LIN {X 0,Y 186.337,Z 566.167,A -85,B 0,C 180,E1 -25155.389,E2 -25155.389} C_VEL
LIN {X 0,Y 191.242,Z 552.199,A -85,B 0,C 180,E1 -25156.919,E2 -25156.919} C_VEL
LIN {X 0,Y 195.713,Z 537.266,A -85,B 0,C 180,E1 -25158.17,E2 -25158.17} C_VEL
LIN {X 0,Y 199.579,Z 520.667,A -85,B 0,C 180,E1 -25159.209,E2 -25159.209} C_VEL
LIN {X 0,Y 202.453,Z 503.675,A -85,B 0,C 180,E1 -25159.932,E2 -25159.932} C_VEL
LIN {X 0,Y 204.963,Z 478.891,A -85,B 0,C 180,E1 -25160.624,E2 -25160.624} C_VEL
LIN {X 0,Y 210.105,Z 419.825,A -85,B 0,C 180,E1 -25162.198,E2 -25162.198} C_VEL
LIN {X 0,Y 205.857,Z 410.908,A -85,B 0,C 180,E1 -25164.939,E2 -25164.939} C_VEL
LIN {X 0,Y 201.466,Z 402.465,A -85,B 0,C 180,E1 -25168.126,E2 -25168.126} C_VEL
LIN {X 0,Y 197.062,Z 394.449,A -85,B 0,C 180,E1 -25171.873,E2 -25171.873} C_VEL
LIN {X 0,Y 194.207,Z 389.891,A -85,B 0,C 180,E1 -25174.726,E2 -25174.726} C_VEL
LIN {X 0,Y 192.533,Z 387.216,A -85,B 0,C 180,E1 -25176.669,E2 -25176.669} C_VEL
LIN {X 0,Y 190.23,Z 383.452,A -85,B 0,C 180,E1 -25179.848,E2 -25179.848} C_VEL
LIN {X 0,Y 188.062,Z 379.924,A -85,B 0,C 180,E1 -25183.828,E2 -25183.828} C_VEL
LIN {X 0,Y 187.657,Z 379.206,A -85,B 0,C 180,E1 -25184.801,E2 -25184.801} C_VEL
LIN {X 0,Y 185.966,Z 376.838,A -85,B 0,C 180,E1 -25192.422,E2 -25192.422} C_VEL
LIN {X 0,Y 186.444,Z 377.313,A -85,B 0,C 180,E1 -25197.839,E2 -25197.839} C_VEL
LIN {X 0,Y 188.185,Z 379.6,A -85,B 0,C 180,E1 -25202.937,E2 -25202.937} C_VEL
LIN {X 0,Y 190.422,Z 383.385,A -85,B 0,C 180,E1 -25207.007,E2 -25207.007} C_VEL
LIN {X 0,Y 193.373,Z 388.362,A -85,B 0,C 180,E1 -25210.924,E2 -25210.924} C_VEL
LIN {X 0,Y 196.208,Z 393.162,A -85,B 0,C 180,E1 -25213.941,E2 -25213.941} C_VEL
LIN {X 0,Y 199.236,Z 398.22,A -85,B 0,C 180,E1 -25216.662,E2 -25216.662} C_VEL
LIN {X 0,Y 203.737,Z 406.658,A -85,B 0,C 180,E1 -25220.178,E2 -25220.178} C_VEL
LIN {X 0,Y 206.831,Z 412.903,A -85,B 0,C 180,E1 -25222.329,E2 -25222.329} C_VEL
LIN {X 0,Y 210.145,Z 421.82,A -85,B 0,C 180,E1 -25224.569,E2 -25224.569} C_VEL
LIN {X 0,Y 202.457,Z 507.175,A -85,B 0,C 180,E1 -25226.824,E2 -25226.824} C_VEL
LIN {X 0,Y 199.785,Z 523.819,A -85,B 0,C 180,E1 -25227.486,E2 -25227.486} C_VEL
LIN {X 0,Y 196.167,Z 539.714,A -85,B 0,C 180,E1 -25228.359,E2 -25228.359} C_VEL
LIN {X 0,Y 191.397,Z 555.971,A -85,B 0,C 180,E1 -25229.566,E2 -25229.566} C_VEL
LIN {X 0,Y 186.522,Z 570.12,A -85,B 0,C 180,E1 -25230.996,E2 -25230.996} C_VEL
LIN {X 0,Y 180.009,Z 585.472,A -85,B 0,C 180,E1 -25232.924,E2 -25232.924} C_VEL
LIN {X 0,Y 177.704,Z 590.398,A -85,B 0,C 180,E1 -25233.681,E2 -25233.681} C_VEL
LIN {X 0,Y 174.983,Z 595.274,A -85,B 0,C 180,E1 -25234.341,E2 -25234.341} C_VEL
LIN {X 0,Y 164.141,Z 608.926,A -85,B 0,C 180,E1 -25235.695,E2 -25235.695} C_VEL
LIN {X 0,Y 160.851,Z 613.295,A -85,B 0,C 180,E1 -25236.464,E2 -25236.464} C_VEL
LIN {X 0,Y 159.931,Z 614.738,A -85,B 0,C 180,E1 -25236.807,E2 -25236.807} C_VEL
LIN {X 0,Y 152.687,Z 626.22,A -85,B 0,C 180,E1 -25240.119,E2 -25240.119} C_VEL
LIN {X 0,Y 144.962,Z 637.569,A -85,B 0,C 180,E1 -25244.349,E2 -25244.349} C_VEL
LIN {X 0,Y 138.444,Z 646.665,A -85,B 0,C 180,E1 -25248.706,E2 -25248.706} C_VEL
LIN {X 0,Y 132.088,Z 655.399,A -85,B 0,C 180,E1 -25254.178,E2 -25254.178} C_VEL
LIN {X 0,Y 126.943,Z 662.627,A -85,B 0,C 180,E1 -25260.115,E2 -25260.115} C_VEL
LIN {X 0,Y 123.111,Z 668.58,A -85,B 0,C 180,E1 -25266.447,E2 -25266.447} C_VEL
LIN {X 0,Y 120.642,Z 673.309,A -85,B 0,C 180,E1 -25273.066,E2 -25273.066} C_VEL
LIN {X 0,Y 119.404,Z 676.892,A -85,B 0,C 180,E1 -25279.83,E2 -25279.83} C_VEL
LIN {X 0,Y 119.27,Z 679.447,A -85,B 0,C 180,E1 -25286.622,E2 -25286.622} C_VEL
LIN {X 0,Y 119.387,Z 680.288,A -85,B 0,C 180,E1 -25290,E2 -25290} C_VEL
LIN {X 0,Y 119.192,Z 681.267,A -85,B 0,C 180,E1 -25296.773,E2 -25296.773} C_VEL
LIN {X 0,Y 119.91,Z 681.236,A -85,B 0,C 180,E1 -25303.559,E2 -25303.559} C_VEL
LIN {X 0,Y 121.953,Z 680.336,A -85,B 0,C 180,E1 -25310.229,E2 -25310.229} C_VEL
LIN {X 0,Y 125.364,Z 678.424,A -85,B 0,C 180,E1 -25316.647,E2 -25316.647} C_VEL
LIN {X 0,Y 130.22,Z 675.643,A -85,B 0,C 180,E1 -25322.664,E2 -25322.664} C_VEL
LIN {X 0,Y 138.009,Z 670.706,A -85,B 0,C 180,E1 -25329.536,E2 -25329.536} C_VEL
LIN {X 0,Y 147.62,Z 664.098,A -85,B 0,C 180,E1 -25335.573,E2 -25335.573} C_VEL
LIN {X 0,Y 156.377,Z 657.468,A -85,B 0,C 180,E1 -25339.821,E2 -25339.821} C_VEL
LIN {X 0,Y 166.999,Z 648.604,A -85,B 0,C 180,E1 -25344.005,E2 -25344.005} C_VEL
LIN {X 0,Y 177.411,Z 638.938,A -85,B 0,C 180,E1 -25347.331,E2 -25347.331} C_VEL
LIN {X 0,Y 186.913,Z 629.099,A -85,B 0,C 180,E1 -25349.861,E2 -25349.861} C_VEL
LIN {X 0,Y 196.077,Z 618.371,A -85,B 0,C 180,E1 -25352.022,E2 -25352.022} C_VEL
LIN {X 0,Y 204.663,Z 607.189,A -85,B 0,C 180,E1 -25353.782,E2 -25353.782} C_VEL
LIN {X 0,Y 213.545,Z 593.939,A -85,B 0,C 180,E1 -25355.391,E2 -25355.391} C_VEL
LIN {X 0,Y 221.834,Z 579.493,A -85,B 0,C 180,E1 -25356.746,E2 -25356.746} C_VEL
LIN {X 0,Y 228.693,Z 565.379,A -85,B 0,C 180,E1 -25357.786,E2 -25357.786} C_VEL
LIN {X 0,Y 234.898,Z 550.175,A -85,B 0,C 180,E1 -25358.63,E2 -25358.63} C_VEL
LIN {X 0,Y 239.98,Z 534.664,A -85,B 0,C 180,E1 -25359.279,E2 -25359.279} C_VEL
LIN {X 0,Y 244.021,Z 518.311,A -85,B 0,C 180,E1 -25359.771,E2 -25359.771} C_VEL
LIN {X 0,Y 246.768,Z 501.84,A -85,B 0,C 180,E1 -25360.179,E2 -25360.179} C_VEL
LIN {X 0,Y 251.671,Z 457.038,A -85,B 0,C 180,E1 -25361.057,E2 -25361.057} C_VEL
LIN {X 0,Y 250.215,Z 453.342,A -85,B 0,C 180,E1 -25363.107,E2 -25363.107} C_VEL
LIN {X 0,Y 248.725,Z 450.046,A -85,B 0,C 180,E1 -25365.709,E2 -25365.709} C_VEL
LIN {X 0,Y 247.616,Z 447.275,A -85,B 0,C 180,E1 -25368.541,E2 -25368.541} C_VEL
LIN {X 0,Y 246.778,Z 445.427,A -85,B 0,C 180,E1 -25373.46,E2 -25373.46} C_VEL
LIN {X 0,Y 247.261,Z 446.348,A -85,B 0,C 180,E1 -25377.569,E2 -25377.569} C_VEL
LIN {X 0,Y 247.838,Z 447.378,A -85,B 0,C 180,E1 -25379.455,E2 -25379.455} C_VEL
LIN {X 0,Y 249.181,Z 450.878,A -85,B 0,C 180,E1 -25382.582,E2 -25382.582} C_VEL
LIN {X 0,Y 250.647,Z 454.357,A -85,B 0,C 180,E1 -25384.977,E2 -25384.977} C_VEL
LIN {X 0,Y 251.649,Z 456.664,A -85,B 0,C 180,E1 -25386.321,E2 -25386.321} C_VEL
LIN {X 0,Y 246.521,Z 502.914,A -85,B 0,C 180,E1 -25387.271,E2 -25387.271} C_VEL
LIN {X 0,Y 243.089,Z 520.449,A -85,B 0,C 180,E1 -25387.703,E2 -25387.703} C_VEL
LIN {X 0,Y 239.582,Z 533.686,A -85,B 0,C 180,E1 -25388.23,E2 -25388.23} C_VEL
LIN {X 0,Y 234.385,Z 549.286,A -85,B 0,C 180,E1 -25389.021,E2 -25389.021} C_VEL
LIN {X 0,Y 228.35,Z 563.869,A -85,B 0,C 180,E1 -25389.976,E2 -25389.976} C_VEL
LIN {X 0,Y 221.177,Z 578.22,A -85,B 0,C 180,E1 -25391.166,E2 -25391.166} C_VEL
LIN {X 0,Y 213.319,Z 591.621,A -85,B 0,C 180,E1 -25392.57,E2 -25392.57} C_VEL
LIN {X 0,Y 204.35,Z 604.831,A -85,B 0,C 180,E1 -25394.347,E2 -25394.347} C_VEL
LIN {X 0,Y 194.601,Z 617.303,A -85,B 0,C 180,E1 -25396.523,E2 -25396.523} C_VEL
LIN {X 0,Y 184.196,Z 628.903,A -85,B 0,C 180,E1 -25399.206,E2 -25399.206} C_VEL
LIN {X 0,Y 174.447,Z 638.43,A -85,B 0,C 180,E1 -25402.087,E2 -25402.087} C_VEL
LIN {X 0,Y 163.931,Z 647.617,A -85,B 0,C 180,E1 -25405.801,E2 -25405.801} C_VEL
LIN {X 0,Y 153.724,Z 655.539,A -85,B 0,C 180,E1 -25410.194,E2 -25410.194} C_VEL
LIN {X 0,Y 145.398,Z 661.433,A -85,B 0,C 180,E1 -25414.742,E2 -25414.742} C_VEL
LIN {X 0,Y 135.919,Z 667.378,A -85,B 0,C 180,E1 -25421.43,E2 -25421.43} C_VEL
LIN {X 0,Y 128.399,Z 671.488,A -85,B 0,C 180,E1 -25428.941,E2 -25428.941} C_VEL
LIN {X 0,Y 123.939,Z 673.501,A -85,B 0,C 180,E1 -25435.455,E2 -25435.455} C_VEL
LIN {X 0,Y 120.965,Z 674.543,A -85,B 0,C 180,E1 -25442.303,E2 -25442.303} C_VEL
LIN {X 0,Y 119.219,Z 674.438,A -85,B 0,C 180,E1 -25450.603,E2 -25450.603} C_VEL
LIN {X 0,Y 118.781,Z 673.527,A -85,B 0,C 180,E1 -25456.309,E2 -25456.309} C_VEL
LIN {X 0,Y 119.189,Z 671.543,A -85,B 0,C 180,E1 -25463.227,E2 -25463.227} C_VEL
LIN {X 0,Y 119.775,Z 670.168,A -85,B 0,C 180,E1 -25466.636,E2 -25466.636} C_VEL
LIN {X 0,Y 121.173,Z 666.756,A -85,B 0,C 180,E1 -25473.325,E2 -25473.325} C_VEL
LIN {X 0,Y 123.801,Z 662.212,A -85,B 0,C 180,E1 -25479.805,E2 -25479.805} C_VEL
LIN {X 0,Y 127.549,Z 656.596,A -85,B 0,C 180,E1 -25485.992,E2 -25485.992} C_VEL
LIN {X 0,Y 132.709,Z 649.749,A -85,B 0,C 180,E1 -25491.759,E2 -25491.759} C_VEL
LIN {X 0,Y 138.915,Z 641.455,A -85,B 0,C 180,E1 -25497.086,E2 -25497.086} C_VEL
LIN {X 0,Y 146.154,Z 631.597,A -85,B 0,C 180,E1 -25501.934,E2 -25501.934} C_VEL
LIN {X 0,Y 153.166,Z 621.472,A -85,B 0,C 180,E1 -25505.805,E2 -25505.805} C_VEL
LIN {X 0,Y 160.611,Z 609.626,A -85,B 0,C 180,E1 -25509.382,E2 -25509.382} C_VEL
LIN {X 0,Y 168.604,Z 595.509,A -85,B 0,C 180,E1 -25512.637,E2 -25512.637} C_VEL
LIN {X 0,Y 175.905,Z 580.954,A -85,B 0,C 180,E1 -25515.167,E2 -25515.167} C_VEL
LIN {X 0,Y 182.102,Z 566.408,A -85,B 0,C 180,E1 -25517.162,E2 -25517.162} C_VEL
LIN {X 0,Y 187.17,Z 552.446,A -85,B 0,C 180,E1 -25518.675,E2 -25518.675} C_VEL
LIN {X 0,Y 191.771,Z 537.524,A -85,B 0,C 180,E1 -25519.909,E2 -25519.909} C_VEL
LIN {X 0,Y 195.744,Z 520.934,A -85,B 0,C 180,E1 -25520.934,E2 -25520.934} C_VEL
LIN {X 0,Y 198.581,Z 504.722,A -85,B 0,C 180,E1 -25521.618,E2 -25521.618} C_VEL
LIN {X 0,Y 201.066,Z 481.743,A -85,B 0,C 180,E1 -25522.255,E2 -25522.255} C_VEL
LIN {X 0,Y 206.306,Z 423.073,A -85,B 0,C 180,E1 -25523.819,E2 -25523.819} C_VEL
LIN {X 0,Y 202.285,Z 414.463,A -85,B 0,C 180,E1 -25526.647,E2 -25526.647} C_VEL
LIN {X 0,Y 198.249,Z 406.566,A -85,B 0,C 180,E1 -25529.852,E2 -25529.852} C_VEL
LIN {X 0,Y 194.814,Z 400.152,A -85,B 0,C 180,E1 -25533.047,E2 -25533.047} C_VEL
LIN {X 0,Y 192.615,Z 396.394,A -85,B 0,C 180,E1 -25535.413,E2 -25535.413} C_VEL
LIN {X 0,Y 190.919,Z 393.617,A -85,B 0,C 180,E1 -25537.498,E2 -25537.498} C_VEL
LIN {X 0,Y 188.925,Z 390.178,A -85,B 0,C 180,E1 -25540.438,E2 -25540.438} C_VEL
LIN {X 0,Y 186.872,Z 386.56,A -85,B 0,C 180,E1 -25544.514,E2 -25544.514} C_VEL
LIN {X 0,Y 185.091,Z 383.896,A -85,B 0,C 180,E1 -25552.386,E2 -25552.386} C_VEL
LIN {X 0,Y 185.392,Z 384.133,A -85,B 0,C 180,E1 -25556.937,E2 -25556.937} C_VEL
LIN {X 0,Y 187.081,Z 386.507,A -85,B 0,C 180,E1 -25562.5,E2 -25562.5} C_VEL
LIN {X 0,Y 189.544,Z 390.974,A -85,B 0,C 180,E1 -25567.122,E2 -25567.122} C_VEL
LIN {X 0,Y 192.144,Z 395.52,A -85,B 0,C 180,E1 -25570.635,E2 -25570.635} C_VEL
LIN {X 0,Y 195.511,Z 401.274,A -85,B 0,C 180,E1 -25574.24,E2 -25574.24} C_VEL
LIN {X 0,Y 199.331,Z 408.496,A -85,B 0,C 180,E1 -25577.653,E2 -25577.653} C_VEL
LIN {X 0,Y 203.777,Z 417.397,A -85,B 0,C 180,E1 -25581.036,E2 -25581.036} C_VEL
LIN {X 0,Y 206.365,Z 424.666,A -85,B 0,C 180,E1 -25582.94,E2 -25582.94} C_VEL
LIN {X 0,Y 198.79,Z 506.406,A -85,B 0,C 180,E1 -25585.08,E2 -25585.08} C_VEL
LIN {X 0,Y 196.258,Z 522.348,A -85,B 0,C 180,E1 -25585.706,E2 -25585.706} C_VEL
LIN {X 0,Y 192.503,Z 538.718,A -85,B 0,C 180,E1 -25586.561,E2 -25586.561} C_VEL
LIN {X 0,Y 187.936,Z 554.142,A -85,B 0,C 180,E1 -25587.649,E2 -25587.649} C_VEL
LIN {X 0,Y 182.881,Z 568.474,A -85,B 0,C 180,E1 -25589.042,E2 -25589.042} C_VEL
LIN {X 0,Y 176.855,Z 582.642,A -85,B 0,C 180,E1 -25590.757,E2 -25590.757} C_VEL
LIN {X 0,Y 170.37,Z 596.075,A -85,B 0,C 180,E1 -25592.856,E2 -25592.856} C_VEL
LIN {X 0,Y 163.617,Z 608.483,A -85,B 0,C 180,E1 -25595.302,E2 -25595.302} C_VEL
LIN {X 0,Y 159.931,Z 614.738,A -85,B 0,C 180,E1 -25596.807,E2 -25596.807} C_VEL
LIN {X 0,Y 156.851,Z 619.027,A -85,B 0,C 180,E1 -25597.773,E2 -25597.773} C_VEL
LIN {X 0,Y 150.414,Z 625.807,A -85,B 0,C 180,E1 -25599.03,E2 -25599.03} C_VEL
LIN {X 0,Y 143.858,Z 632.213,A -85,B 0,C 180,E1 -25600.51,E2 -25600.51} C_VEL
LIN {X 0,Y 140.658,Z 635.915,A -85,B 0,C 180,E1 -25601.842,E2 -25601.842} C_VEL
LIN {X 0,Y 133.09,Z 645.985,A -85,B 0,C 180,E1 -25606.648,E2 -25606.648} C_VEL
LIN {X 0,Y 126.297,Z 654.778,A -85,B 0,C 180,E1 -25612.258,E2 -25612.258} C_VEL
LIN {X 0,Y 120.715,Z 662.087,A -85,B 0,C 180,E1 -25618.401,E2 -25618.401} C_VEL
LIN {X 0,Y 116.516,Z 668.116,A -85,B 0,C 180,E1 -25625.025,E2 -25625.025} C_VEL
LIN {X 0,Y 113.799,Z 672.884,A -85,B 0,C 180,E1 -25632.014,E2 -25632.014} C_VEL
LIN {X 0,Y 112.374,Z 676.537,A -85,B 0,C 180,E1 -25639.186,E2 -25639.186} C_VEL
LIN {X 0,Y 112.155,Z 679.126,A -85,B 0,C 180,E1 -25646.408,E2 -25646.408} C_VEL
LIN {X 0,Y 112.297,Z 680.001,A -85,B 0,C 180,E1 -25650,E2 -25650} C_VEL
LIN {X 0,Y 112.111,Z 681.043,A -85,B 0,C 180,E1 -25657.203,E2 -25657.203} C_VEL
LIN {X 0,Y 112.957,Z 681.043,A -85,B 0,C 180,E1 -25664.411,E2 -25664.411} C_VEL
LIN {X 0,Y 115.228,Z 680.198,A -85,B 0,C 180,E1 -25671.467,E2 -25671.467} C_VEL
LIN {X 0,Y 118.989,Z 678.327,A -85,B 0,C 180,E1 -25678.198,E2 -25678.198} C_VEL
LIN {X 0,Y 124.235,Z 675.596,A -85,B 0,C 180,E1 -25684.451,E2 -25684.451} C_VEL
LIN {X 0,Y 132.542,Z 670.71,A -85,B 0,C 180,E1 -25691.515,E2 -25691.515} C_VEL
LIN {X 0,Y 140.542,Z 665.601,A -85,B 0,C 180,E1 -25696.477,E2 -25696.477} C_VEL
LIN {X 0,Y 149.486,Z 659.434,A -85,B 0,C 180,E1 -25700.873,E2 -25700.873} C_VEL
LIN {X 0,Y 160.12,Z 651.186,A -85,B 0,C 180,E1 -25705.085,E2 -25705.085} C_VEL
LIN {X 0,Y 170.974,Z 641.786,A -85,B 0,C 180,E1 -25708.534,E2 -25708.534} C_VEL
LIN {X 0,Y 180.621,Z 632.46,A -85,B 0,C 180,E1 -25711.103,E2 -25711.103} C_VEL
LIN {X 0,Y 190.392,Z 621.889,A -85,B 0,C 180,E1 -25713.333,E2 -25713.333} C_VEL
LIN {X 0,Y 199.233,Z 610.945,A -85,B 0,C 180,E1 -25715.157,E2 -25715.157} C_VEL
LIN {X 0,Y 208.441,Z 598.186,A -85,B 0,C 180,E1 -25716.75,E2 -25716.75} C_VEL
LIN {X 0,Y 215.328,Z 587.258,A -85,B 0,C 180,E1 -25717.839,E2 -25717.839} C_VEL
LIN {X 0,Y 223.015,Z 573.084,A -85,B 0,C 180,E1 -25719.003,E2 -25719.003} C_VEL
LIN {X 0,Y 230.073,Z 557.669,A -85,B 0,C 180,E1 -25719.937,E2 -25719.937} C_VEL
LIN {X 0,Y 236.002,Z 541.731,A -85,B 0,C 180,E1 -25720.672,E2 -25720.672} C_VEL
LIN {X 0,Y 240.871,Z 524.827,A -85,B 0,C 180,E1 -25721.226,E2 -25721.226} C_VEL
LIN {X 0,Y 244.355,Z 507.541,A -85,B 0,C 180,E1 -25721.647,E2 -25721.647} C_VEL
LIN {X 0,Y 247.772,Z 478.748,A -85,B 0,C 180,E1 -25722.229,E2 -25722.229} C_VEL
LIN {X 0,Y 249.613,Z 461.626,A -85,B 0,C 180,E1 -25722.593,E2 -25722.593} C_VEL
LIN {X 0,Y 247.851,Z 457.249,A -85,B 0,C 180,E1 -25725.657,E2 -25725.657} C_VEL
LIN {X 0,Y 246.669,Z 454.257,A -85,B 0,C 180,E1 -25728.732,E2 -25728.732} C_VEL
LIN {X 0,Y 245.902,Z 452.486,A -85,B 0,C 180,E1 -25733.436,E2 -25733.436} C_VEL
LIN {X 0,Y 246.355,Z 453.369,A -85,B 0,C 180,E1 -25737.466,E2 -25737.466} C_VEL
LIN {X 0,Y 246.863,Z 454.409,A -85,B 0,C 180,E1 -25739.233,E2 -25739.233} C_VEL
LIN {X 0,Y 248.064,Z 457.689,A -85,B 0,C 180,E1 -25742.201,E2 -25742.201} C_VEL
LIN {X 0,Y 249.592,Z 461.539,A -85,B 0,C 180,E1 -25744.816,E2 -25744.816} C_VEL
LIN {X 0,Y 244.9,Z 502.927,A -85,B 0,C 180,E1 -25745.656,E2 -25745.656} C_VEL
LIN {X 0,Y 241.502,Z 520.151,A -85,B 0,C 180,E1 -25746.059,E2 -25746.059} C_VEL
LIN {X 0,Y 237.961,Z 533.436,A -85,B 0,C 180,E1 -25746.56,E2 -25746.56} C_VEL
LIN {X 0,Y 232.923,Z 548.501,A -85,B 0,C 180,E1 -25747.278,E2 -25747.278} C_VEL
LIN {X 0,Y 227.178,Z 562.272,A -85,B 0,C 180,E1 -25748.125,E2 -25748.125} C_VEL
LIN {X 0,Y 220.445,Z 575.904,A -85,B 0,C 180,E1 -25749.173,E2 -25749.173} C_VEL
LIN {X 0,Y 212.625,Z 589.418,A -85,B 0,C 180,E1 -25750.471,E2 -25750.471} C_VEL
LIN {X 0,Y 203.251,Z 603.217,A -85,B 0,C 180,E1 -25752.199,E2 -25752.199} C_VEL
LIN {X 0,Y 193.847,Z 615.115,A -85,B 0,C 180,E1 -25754.11,E2 -25754.11} C_VEL
LIN {X 0,Y 183.317,Z 626.81,A -85,B 0,C 180,E1 -25756.573,E2 -25756.573} C_VEL
LIN {X 0,Y 173.548,Z 636.396,A -85,B 0,C 180,E1 -25759.222,E2 -25759.222} C_VEL
LIN {X 0,Y 163.631,Z 645.048,A -85,B 0,C 180,E1 -25762.376,E2 -25762.376} C_VEL
LIN {X 0,Y 152.998,Z 653.212,A -85,B 0,C 180,E1 -25766.396,E2 -25766.396} C_VEL
LIN {X 0,Y 143.431,Z 659.807,A -85,B 0,C 180,E1 -25770.964,E2 -25770.964} C_VEL
LIN {X 0,Y 134.884,Z 665.136,A -85,B 0,C 180,E1 -25776.136,E2 -25776.136} C_VEL
LIN {X 0,Y 128.438,Z 668.668,A -85,B 0,C 180,E1 -25781.046,E2 -25781.046} C_VEL
LIN {X 0,Y 122.767,Z 671.515,A -85,B 0,C 180,E1 -25786.61,E2 -25786.61} C_VEL
LIN {X 0,Y 117.792,Z 673.612,A -85,B 0,C 180,E1 -25793.369,E2 -25793.369} C_VEL
LIN {X 0,Y 114.371,Z 674.737,A -85,B 0,C 180,E1 -25800.554,E2 -25800.554} C_VEL
LIN {X 0,Y 112.169,Z 674.634,A -85,B 0,C 180,E1 -25810.03,E2 -25810.03} C_VEL
LIN {X 0,Y 111.716,Z 673.844,A -85,B 0,C 180,E1 -25815.425,E2 -25815.425} C_VEL
LIN {X 0,Y 112.014,Z 671.899,A -85,B 0,C 180,E1 -25822.791,E2 -25822.791} C_VEL
LIN {X 0,Y 112.663,Z 670.532,A -85,B 0,C 180,E1 -25826.495,E2 -25826.495} C_VEL
LIN {X 0,Y 114.07,Z 667.22,A -85,B 0,C 180,E1 -25833.532,E2 -25833.532} C_VEL
LIN {X 0,Y 116.812,Z 662.735,A -85,B 0,C 180,E1 -25840.398,E2 -25840.398} C_VEL
LIN {X 0,Y 120.751,Z 657.213,A -85,B 0,C 180,E1 -25846.918,E2 -25846.918} C_VEL
LIN {X 0,Y 126.15,Z 650.416,A -85,B 0,C 180,E1 -25852.953,E2 -25852.953} C_VEL
LIN {X 0,Y 132.658,Z 642.229,A -85,B 0,C 180,E1 -25858.477,E2 -25858.477} C_VEL
LIN {X 0,Y 140.211,Z 632.49,A -85,B 0,C 180,E1 -25863.461,E2 -25863.461} C_VEL
LIN {X 0,Y 147.514,Z 622.5,A -85,B 0,C 180,E1 -25867.405,E2 -25867.405} C_VEL
LIN {X 0,Y 155.241,Z 610.736,A -85,B 0,C 180,E1 -25871.028,E2 -25871.028} C_VEL
LIN {X 0,Y 162.907,Z 597.852,A -85,B 0,C 180,E1 -25874.079,E2 -25874.079} C_VEL
LIN {X 0,Y 169.725,Z 585.031,A -85,B 0,C 180,E1 -25876.439,E2 -25876.439} C_VEL
LIN {X 0,Y 176.143,Z 571.324,A -85,B 0,C 180,E1 -25878.427,E2 -25878.427} C_VEL
LIN {X 0,Y 181.956,Z 556.504,A -85,B 0,C 180,E1 -25880.144,E2 -25880.144} C_VEL
LIN {X 0,Y 186.973,Z 541.204,A -85,B 0,C 180,E1 -25881.472,E2 -25881.472} C_VEL
LIN {X 0,Y 191.227,Z 524.964,A -85,B 0,C 180,E1 -25882.524,E2 -25882.524} C_VEL
LIN {X 0,Y 194.536,Z 508.056,A -85,B 0,C 180,E1 -25883.287,E2 -25883.287} C_VEL
LIN {X 0,Y 196.755,Z 490.477,A -85,B 0,C 180,E1 -25883.816,E2 -25883.816} C_VEL
LIN {X 0,Y 202.665,Z 426.35,A -85,B 0,C 180,E1 -25885.498,E2 -25885.498} C_VEL
LIN {X 0,Y 198.551,Z 417.45,A -85,B 0,C 180,E1 -25888.675,E2 -25888.675} C_VEL
LIN {X 0,Y 194.579,Z 409.447,A -85,B 0,C 180,E1 -25892.249,E2 -25892.249} C_VEL
LIN {X 0,Y 191.743,Z 404.049,A -85,B 0,C 180,E1 -25895.294,E2 -25895.294} C_VEL
LIN {X 0,Y 189.57,Z 400.362,A -85,B 0,C 180,E1 -25898.031,E2 -25898.031} C_VEL
LIN {X 0,Y 187.572,Z 396.83,A -85,B 0,C 180,E1 -25901.146,E2 -25901.146} C_VEL
LIN {X 0,Y 185.658,Z 393.172,A -85,B 0,C 180,E1 -25905.328,E2 -25905.328} C_VEL
LIN {X 0,Y 184.207,Z 390.89,A -85,B 0,C 180,E1 -25912.733,E2 -25912.733} C_VEL
LIN {X 0,Y 184.675,Z 391.457,A -85,B 0,C 180,E1 -25917.818,E2 -25917.818} C_VEL
LIN {X 0,Y 185.989,Z 393.414,A -85,B 0,C 180,E1 -25922.059,E2 -25922.059} C_VEL
LIN {X 0,Y 188.27,Z 397.752,A -85,B 0,C 180,E1 -25926.593,E2 -25926.593} C_VEL
LIN {X 0,Y 190.617,Z 402.069,A -85,B 0,C 180,E1 -25929.951,E2 -25929.951} C_VEL
LIN {X 0,Y 193.683,Z 407.582,A -85,B 0,C 180,E1 -25933.441,E2 -25933.441} C_VEL
LIN {X 0,Y 197.536,Z 415.227,A -85,B 0,C 180,E1 -25937.068,E2 -25937.068} C_VEL
LIN {X 0,Y 201.247,Z 423.14,A -85,B 0,C 180,E1 -25940.059,E2 -25940.059} C_VEL
LIN {X 0,Y 202.728,Z 427.476,A -85,B 0,C 180,E1 -25941.233,E2 -25941.233} C_VEL
LIN {X 0,Y 195.206,Z 506.669,A -85,B 0,C 180,E1 -25943.307,E2 -25943.307} C_VEL
LIN {X 0,Y 192.434,Z 523.206,A -85,B 0,C 180,E1 -25943.942,E2 -25943.942} C_VEL
LIN {X 0,Y 188.664,Z 539.033,A -85,B 0,C 180,E1 -25944.77,E2 -25944.77} C_VEL
LIN {X 0,Y 183.62,Z 555.34,A -85,B 0,C 180,E1 -25945.914,E2 -25945.914} C_VEL
LIN {X 0,Y 178.126,Z 570.361,A -85,B 0,C 180,E1 -25947.409,E2 -25947.409} C_VEL
LIN {X 0,Y 171.237,Z 585.631,A -85,B 0,C 180,E1 -25949.291,E2 -25949.291} C_VEL
LIN {X 0,Y 164.032,Z 599.605,A -85,B 0,C 180,E1 -25951.62,E2 -25951.62} C_VEL
LIN {X 0,Y 157.07,Z 611.502,A -85,B 0,C 180,E1 -25954.13,E2 -25954.13} C_VEL
LIN {X 0,Y 149.036,Z 624.035,A -85,B 0,C 180,E1 -25957.56,E2 -25957.56} C_VEL
LIN {X 0,Y 141.029,Z 635.415,A -85,B 0,C 180,E1 -25961.626,E2 -25961.626} C_VEL
LIN {X 0,Y 140.658,Z 635.915,A -85,B 0,C 180,E1 -25961.842,E2 -25961.842} C_VEL
LIN {X 0,Y 137.48,Z 639.567,A -85,B 0,C 180,E1 -25963.273,E2 -25963.273} C_VEL
LIN {X 0,Y 130.869,Z 645.179,A -85,B 0,C 180,E1 -25965.331,E2 -25965.331} C_VEL
LIN {X 0,Y 124.298,Z 650.411,A -85,B 0,C 180,E1 -25967.689,E2 -25967.689} C_VEL
LIN {X 0,Y 121.275,Z 653.383,A -85,B 0,C 180,E1 -25969.588,E2 -25969.588} C_VEL
LIN {X 0,Y 114.621,Z 661.548,A -85,B 0,C 180,E1 -25976.507,E2 -25976.507} C_VEL
LIN {X 0,Y 110.002,Z 667.651,A -85,B 0,C 180,E1 -25983.434,E2 -25983.434} C_VEL
LIN {X 0,Y 106.969,Z 672.457,A -85,B 0,C 180,E1 -25990.822,E2 -25990.822} C_VEL
LIN {X 0,Y 105.338,Z 676.181,A -85,B 0,C 180,E1 -25998.454,E2 -25998.454} C_VEL
LIN {X 0,Y 105.068,Z 678.806,A -85,B 0,C 180,E1 -26006.165,E2 -26006.165} C_VEL
LIN {X 0,Y 105.214,Z 679.714,A -85,B 0,C 180,E1 -26010,E2 -26010} C_VEL
LIN {X 0,Y 105.035,Z 680.805,A -85,B 0,C 180,E1 -26017.691,E2 -26017.691} C_VEL
LIN {X 0,Y 106.017,Z 680.849,A -85,B 0,C 180,E1 -26025.377,E2 -26025.377} C_VEL
LIN {X 0,Y 108.563,Z 680.04,A -85,B 0,C 180,E1 -26032.857,E2 -26032.857} C_VEL
LIN {X 0,Y 112.703,Z 678.23,A -85,B 0,C 180,E1 -26039.926,E2 -26039.926} C_VEL
LIN {X 0,Y 118.377,Z 675.533,A -85,B 0,C 180,E1 -26046.42,E2 -26046.42} C_VEL
LIN {X 0,Y 127.25,Z 670.722,A -85,B 0,C 180,E1 -26053.66,E2 -26053.66} C_VEL
LIN {X 0,Y 135.695,Z 665.695,A -85,B 0,C 180,E1 -26058.677,E2 -26058.677} C_VEL
LIN {X 0,Y 145.083,Z 659.578,A -85,B 0,C 180,E1 -26063.062,E2 -26063.062} C_VEL
LIN {X 0,Y 156.98,Z 650.774,A -85,B 0,C 180,E1 -26067.506,E2 -26067.506} C_VEL
LIN {X 0,Y 167.367,Z 642.098,A -85,B 0,C 180,E1 -26070.614,E2 -26070.614} C_VEL
LIN {X 0,Y 177.301,Z 632.878,A -85,B 0,C 180,E1 -26073.11,E2 -26073.11} C_VEL
LIN {X 0,Y 188.47,Z 621.091,A -85,B 0,C 180,E1 -26075.515,E2 -26075.515} C_VEL
LIN {X 0,Y 198.064,Z 609.43,A -85,B 0,C 180,E1 -26077.306,E2 -26077.306} C_VEL
LIN {X 0,Y 206.549,Z 597.799,A -85,B 0,C 180,E1 -26078.664,E2 -26078.664} C_VEL
LIN {X 0,Y 215.096,Z 584.28,A -85,B 0,C 180,E1 -26079.947,E2 -26079.947} C_VEL
LIN {X 0,Y 222.979,Z 569.514,A -85,B 0,C 180,E1 -26081.008,E2 -26081.008} C_VEL
LIN {X 0,Y 229.358,Z 555.21,A -85,B 0,C 180,E1 -26081.788,E2 -26081.788} C_VEL
LIN {X 0,Y 234.994,Z 539.847,A -85,B 0,C 180,E1 -26082.42,E2 -26082.42} C_VEL
LIN {X 0,Y 239.539,Z 524.02,A -85,B 0,C 180,E1 -26082.906,E2 -26082.906} C_VEL
LIN {X 0,Y 242.862,Z 507.698,A -85,B 0,C 180,E1 -26083.284,E2 -26083.284} C_VEL
LIN {X 0,Y 246.443,Z 478.413,A -85,B 0,C 180,E1 -26083.851,E2 -26083.851} C_VEL
LIN {X 0,Y 247.751,Z 466.716,A -85,B 0,C 180,E1 -26084.076,E2 -26084.076} C_VEL
LIN {X 0,Y 246.528,Z 463.62,A -85,B 0,C 180,E1 -26086.545,E2 -26086.545} C_VEL
LIN {X 0,Y 245.723,Z 461.251,A -85,B 0,C 180,E1 -26088.925,E2 -26088.925} C_VEL
LIN {X 0,Y 245.026,Z 459.546,A -85,B 0,C 180,E1 -26093.413,E2 -26093.413} C_VEL
LIN {X 0,Y 245.431,Z 460.369,A -85,B 0,C 180,E1 -26097.281,E2 -26097.281} C_VEL
LIN {X 0,Y 245.875,Z 461.319,A -85,B 0,C 180,E1 -26098.931,E2 -26098.931} C_VEL
LIN {X 0,Y 246.973,Z 464.554,A -85,B 0,C 180,E1 -26101.849,E2 -26101.849} C_VEL
LIN {X 0,Y 247.735,Z 466.47,A -85,B 0,C 180,E1 -26103.304,E2 -26103.304} C_VEL
LIN {X 0,Y 243.322,Z 503.908,A -85,B 0,C 180,E1 -26104.043,E2 -26104.043} C_VEL
LIN {X 0,Y 239.879,Z 520.923,A -85,B 0,C 180,E1 -26104.427,E2 -26104.427} C_VEL
LIN {X 0,Y 236.032,Z 534.848,A -85,B 0,C 180,E1 -26104.941,E2 -26104.941} C_VEL
LIN {X 0,Y 230.424,Z 550.821,A -85,B 0,C 180,E1 -26105.688,E2 -26105.688} C_VEL
LIN {X 0,Y 225.415,Z 562.517,A -85,B 0,C 180,E1 -26106.38,E2 -26106.38} C_VEL
LIN {X 0,Y 217.937,Z 577.251,A -85,B 0,C 180,E1 -26107.469,E2 -26107.469} C_VEL
LIN {X 0,Y 209.765,Z 590.864,A -85,B 0,C 180,E1 -26108.744,E2 -26108.744} C_VEL
LIN {X 0,Y 200.091,Z 604.635,A -85,B 0,C 180,E1 -26110.43,E2 -26110.43} C_VEL
LIN {X 0,Y 190.592,Z 616.259,A -85,B 0,C 180,E1 -26112.263,E2 -26112.263} C_VEL
LIN {X 0,Y 181.321,Z 626.261,A -85,B 0,C 180,E1 -26114.302,E2 -26114.302} C_VEL
LIN {X 0,Y 171.302,Z 635.908,A -85,B 0,C 180,E1 -26116.825,E2 -26116.825} C_VEL
LIN {X 0,Y 160.747,Z 644.824,A -85,B 0,C 180,E1 -26119.948,E2 -26119.948} C_VEL
LIN {X 0,Y 149.79,Z 652.962,A -85,B 0,C 180,E1 -26123.805,E2 -26123.805} C_VEL
LIN {X 0,Y 139.676,Z 659.656,A -85,B 0,C 180,E1 -26128.292,E2 -26128.292} C_VEL
LIN {X 0,Y 130.541,Z 665.057,A -85,B 0,C 180,E1 -26133.437,E2 -26133.437} C_VEL
LIN {X 0,Y 120.724,Z 670.064,A -85,B 0,C 180,E1 -26140.816,E2 -26140.816} C_VEL
LIN {X 0,Y 114.426,Z 672.754,A -85,B 0,C 180,E1 -26147.497,E2 -26147.497} C_VEL
LIN {X 0,Y 109.655,Z 674.449,A -85,B 0,C 180,E1 -26154.772,E2 -26154.772} C_VEL
LIN {X 0,Y 106.52,Z 675.061,A -85,B 0,C 180,E1 -26162.493,E2 -26162.493} C_VEL
LIN {X 0,Y 105.019,Z 674.685,A -85,B 0,C 180,E1 -26170.451,E2 -26170.451} C_VEL
LIN {X 0,Y 104.586,Z 673.323,A -85,B 0,C 180,E1 -26178.369,E2 -26178.369} C_VEL
LIN {X 0,Y 105.591,Z 670.729,A -85,B 0,C 180,E1 -26186.774,E2 -26186.774} C_VEL
LIN {X 0,Y 106.971,Z 667.658,A -85,B 0,C 180,E1 -26193.767,E2 -26193.767} C_VEL
LIN {X 0,Y 109.842,Z 663.258,A -85,B 0,C 180,E1 -26201.066,E2 -26201.066} C_VEL
LIN {X 0,Y 113.988,Z 657.83,A -85,B 0,C 180,E1 -26207.955,E2 -26207.955} C_VEL
LIN {X 0,Y 119.653,Z 651.083,A -85,B 0,C 180,E1 -26214.277,E2 -26214.277} C_VEL
LIN {X 0,Y 126.49,Z 643.002,A -85,B 0,C 180,E1 -26220.003,E2 -26220.003} C_VEL
LIN {X 0,Y 134.378,Z 633.383,A -85,B 0,C 180,E1 -26225.121,E2 -26225.121} C_VEL
LIN {X 0,Y 141.972,Z 623.484,A -85,B 0,C 180,E1 -26229.135,E2 -26229.135} C_VEL
LIN {X 0,Y 150.008,Z 611.842,A -85,B 0,C 180,E1 -26232.791,E2 -26232.791} C_VEL
LIN {X 0,Y 157.938,Z 599.137,A -85,B 0,C 180,E1 -26235.851,E2 -26235.851} C_VEL
LIN {X 0,Y 165.616,Z 585.262,A -85,B 0,C 180,E1 -26238.411,E2 -26238.411} C_VEL
LIN {X 0,Y 172.228,Z 571.564,A -85,B 0,C 180,E1 -26240.373,E2 -26240.373} C_VEL
LIN {X 0,Y 178.225,Z 556.736,A -85,B 0,C 180,E1 -26242.061,E2 -26242.061} C_VEL
LIN {X 0,Y 183.381,Z 541.432,A -85,B 0,C 180,E1 -26243.362,E2 -26243.362} C_VEL
LIN {X 0,Y 187.75,Z 525.183,A -85,B 0,C 180,E1 -26244.389,E2 -26244.389} C_VEL
LIN {X 0,Y 190.998,Z 509.103,A -85,B 0,C 180,E1 -26245.11,E2 -26245.11} C_VEL
LIN {X 0,Y 193.3,Z 491.834,A -85,B 0,C 180,E1 -26245.624,E2 -26245.624} C_VEL
LIN {X 0,Y 199.205,Z 429.792,A -85,B 0,C 180,E1 -26247.217,E2 -26247.217} C_VEL
LIN {X 0,Y 195.415,Z 421.364,A -85,B 0,C 180,E1 -26250.437,E2 -26250.437} C_VEL
LIN {X 0,Y 191.659,Z 413.463,A -85,B 0,C 180,E1 -26254.242,E2 -26254.242} C_VEL
LIN {X 0,Y 189.113,Z 408.675,A -85,B 0,C 180,E1 -26257.35,E2 -26257.35} C_VEL
LIN {X 0,Y 186.432,Z 403.709,A -85,B 0,C 180,E1 -26261.54,E2 -26261.54} C_VEL
LIN {X 0,Y 184.536,Z 400.057,A -85,B 0,C 180,E1 -26265.934,E2 -26265.934} C_VEL
LIN {X 0,Y 183.339,Z 397.998,A -85,B 0,C 180,E1 -26272.386,E2 -26272.386} C_VEL
LIN {X 0,Y 183.629,Z 398.243,A -85,B 0,C 180,E1 -26276.907,E2 -26276.907} C_VEL
LIN {X 0,Y 184.886,Z 400.228,A -85,B 0,C 180,E1 -26281.541,E2 -26281.541} C_VEL
LIN {X 0,Y 186.957,Z 404.447,A -85,B 0,C 180,E1 -26285.966,E2 -26285.966} C_VEL
LIN {X 0,Y 189.07,Z 408.538,A -85,B 0,C 180,E1 -26289.198,E2 -26289.198} C_VEL
LIN {X 0,Y 191.95,Z 414.018,A -85,B 0,C 180,E1 -26292.689,E2 -26292.689} C_VEL
LIN {X 0,Y 195.459,Z 421.346,A -85,B 0,C 180,E1 -26296.203,E2 -26296.203} C_VEL
LIN {X 0,Y 198.809,Z 428.959,A -85,B 0,C 180,E1 -26299.086,E2 -26299.086} C_VEL
LIN {X 0,Y 199.316,Z 430.45,A -85,B 0,C 180,E1 -26299.517,E2 -26299.517} C_VEL
LIN {X 0,Y 191.852,Z 506.478,A -85,B 0,C 180,E1 -26301.454,E2 -26301.454} C_VEL
LIN {X 0,Y 189.112,Z 522.617,A -85,B 0,C 180,E1 -26302.066,E2 -26302.066} C_VEL
LIN {X 0,Y 185.023,Z 539.347,A -85,B 0,C 180,E1 -26302.91,E2 -26302.91} C_VEL
LIN {X 0,Y 179.857,Z 555.535,A -85,B 0,C 180,E1 -26304.022,E2 -26304.022} C_VEL
LIN {X 0,Y 174.209,Z 570.476,A -85,B 0,C 180,E1 -26305.49,E2 -26305.49} C_VEL
LIN {X 0,Y 167.129,Z 585.705,A -85,B 0,C 180,E1 -26307.336,E2 -26307.336} C_VEL
LIN {X 0,Y 159.686,Z 599.635,A -85,B 0,C 180,E1 -26309.632,E2 -26309.632} C_VEL
LIN {X 0,Y 151.839,Z 612.488,A -85,B 0,C 180,E1 -26312.359,E2 -26312.359} C_VEL
LIN {X 0,Y 143.435,Z 624.949,A -85,B 0,C 180,E1 -26315.855,E2 -26315.855} C_VEL
LIN {X 0,Y 135.097,Z 636.201,A -85,B 0,C 180,E1 -26320.021,E2 -26320.021} C_VEL
LIN {X 0,Y 126.944,Z 646.477,A -85,B 0,C 180,E1 -26325.1,E2 -26325.1} C_VEL
LIN {X 0,Y 121.275,Z 653.383,A -85,B 0,C 180,E1 -26329.588,E2 -26329.588} C_VEL
LIN {X 0,Y 118.349,Z 656.286,A -85,B 0,C 180,E1 -26331.627,E2 -26331.627} C_VEL
LIN {X 0,Y 107.336,Z 663.847,A -85,B 0,C 180,E1 -26337.686,E2 -26337.686} C_VEL
LIN {X 0,Y 104.532,Z 666.056,A -85,B 0,C 180,E1 -26340.226,E2 -26340.226} C_VEL
LIN {X 0,Y 103.88,Z 666.792,A -85,B 0,C 180,E1 -26341.162,E2 -26341.162} C_VEL
LIN {X 0,Y 100.202,Z 672.031,A -85,B 0,C 180,E1 -26349.471,E2 -26349.471} C_VEL
LIN {X 0,Y 98.334,Z 675.826,A -85,B 0,C 180,E1 -26357.619,E2 -26357.619} C_VEL
LIN {X 0,Y 97.951,Z 678.484,A -85,B 0,C 180,E1 -26365.886,E2 -26365.886} C_VEL
LIN {X 0,Y 98.131,Z 679.427,A -85,B 0,C 180,E1 -26370,E2 -26370} C_VEL
LIN {X 0,Y 97.981,Z 680.551,A -85,B 0,C 180,E1 -26378.248,E2 -26378.248} C_VEL
LIN {X 0,Y 99.115,Z 680.655,A -85,B 0,C 180,E1 -26386.478,E2 -26386.478} C_VEL
LIN {X 0,Y 101.974,Z 679.878,A -85,B 0,C 180,E1 -26394.427,E2 -26394.427} C_VEL
LIN {X 0,Y 106.538,Z 678.135,A -85,B 0,C 180,E1 -26401.853,E2 -26401.853} C_VEL
LIN {X 0,Y 112.658,Z 675.477,A -85,B 0,C 180,E1 -26408.597,E2 -26408.597} C_VEL
LIN {X 0,Y 122.005,Z 670.81,A -85,B 0,C 180,E1 -26415.903,E2 -26415.903} C_VEL
LIN {X 0,Y 131.075,Z 665.788,A -85,B 0,C 180,E1 -26421.03,E2 -26421.03} C_VEL
LIN {X 0,Y 140.911,Z 659.71,A -85,B 0,C 180,E1 -26425.381,E2 -26425.381} C_VEL
LIN {X 0,Y 152.75,Z 651.367,A -85,B 0,C 180,E1 -26429.597,E2 -26429.597} C_VEL
LIN {X 0,Y 163.988,Z 642.411,A -85,B 0,C 180,E1 -26432.784,E2 -26432.784} C_VEL
LIN {X 0,Y 174.208,Z 633.294,A -85,B 0,C 180,E1 -26435.191,E2 -26435.191} C_VEL
LIN {X 0,Y 185.515,Z 621.722,A -85,B 0,C 180,E1 -26437.478,E2 -26437.478} C_VEL
LIN {X 0,Y 195.45,Z 610.041,A -85,B 0,C 180,E1 -26439.215,E2 -26439.215} C_VEL
LIN {X 0,Y 204.877,Z 597.417,A -85,B 0,C 180,E1 -26440.622,E2 -26440.622} C_VEL
LIN {X 0,Y 212.786,Z 585.19,A -85,B 0,C 180,E1 -26441.727,E2 -26441.727} C_VEL
LIN {X 0,Y 220.797,Z 570.628,A -85,B 0,C 180,E1 -26442.729,E2 -26442.729} C_VEL
LIN {X 0,Y 227.266,Z 556.68,A -85,B 0,C 180,E1 -26443.466,E2 -26443.466} C_VEL
LIN {X 0,Y 232.979,Z 541.85,A -85,B 0,C 180,E1 -26444.058,E2 -26444.058} C_VEL
LIN {X 0,Y 237.915,Z 525.281,A -85,B 0,C 180,E1 -26444.547,E2 -26444.547} C_VEL
LIN {X 0,Y 241.511,Z 508.364,A -85,B 0,C 180,E1 -26444.925,E2 -26444.925} C_VEL
LIN {X 0,Y 244.503,Z 485.419,A -85,B 0,C 180,E1 -26445.356,E2 -26445.356} C_VEL
LIN {X 0,Y 246.016,Z 472.03,A -85,B 0,C 180,E1 -26445.622,E2 -26445.622} C_VEL
LIN {X 0,Y 245.384,Z 470.269,A -85,B 0,C 180,E1 -26447.132,E2 -26447.132} C_VEL
LIN {X 0,Y 244.711,Z 468.153,A -85,B 0,C 180,E1 -26449.353,E2 -26449.353} C_VEL
LIN {X 0,Y 244.15,Z 466.597,A -85,B 0,C 180,E1 -26453.389,E2 -26453.389} C_VEL
LIN {X 0,Y 244.514,Z 467.375,A -85,B 0,C 180,E1 -26457.118,E2 -26457.118} C_VEL
LIN {X 0,Y 244.919,Z 468.344,A -85,B 0,C 180,E1 -26458.732,E2 -26458.732} C_VEL
LIN {X 0,Y 245.875,Z 471.351,A -85,B 0,C 180,E1 -26461.447,E2 -26461.447} C_VEL
LIN {X 0,Y 246.025,Z 471.82,A -85,B 0,C 180,E1 -26461.791,E2 -26461.791} C_VEL
LIN {X 0,Y 242.053,Z 504.404,A -85,B 0,C 180,E1 -26462.401,E2 -26462.401} C_VEL
LIN {X 0,Y 238.354,Z 522.193,A -85,B 0,C 180,E1 -26462.779,E2 -26462.779} C_VEL
LIN {X 0,Y 234.373,Z 536.087,A -85,B 0,C 180,E1 -26463.288,E2 -26463.288} C_VEL
LIN {X 0,Y 228.53,Z 552.137,A -85,B 0,C 180,E1 -26464.006,E2 -26464.006} C_VEL
LIN {X 0,Y 223.021,Z 564.616,A -85,B 0,C 180,E1 -26464.729,E2 -26464.729} C_VEL
LIN {X 0,Y 215.569,Z 578.71,A -85,B 0,C 180,E1 -26465.743,E2 -26465.743} C_VEL
LIN {X 0,Y 207.104,Z 592.312,A -85,B 0,C 180,E1 -26466.977,E2 -26466.977} C_VEL
LIN {X 0,Y 198.059,Z 604.861,A -85,B 0,C 180,E1 -26468.455,E2 -26468.455} C_VEL
LIN {X 0,Y 187.538,Z 617.404,A -85,B 0,C 180,E1 -26470.351,E2 -26470.351} C_VEL
LIN {X 0,Y 176.477,Z 628.785,A -85,B 0,C 180,E1 -26472.659,E2 -26472.659} C_VEL
LIN {X 0,Y 165.748,Z 638.444,A -85,B 0,C 180,E1 -26475.281,E2 -26475.281} C_VEL
LIN {X 0,Y 154.38,Z 647.451,A -85,B 0,C 180,E1 -26478.584,E2 -26478.584} C_VEL
LIN {X 0,Y 144.158,Z 654.573,A -85,B 0,C 180,E1 -26482.136,E2 -26482.136} C_VEL
LIN {X 0,Y 133.717,Z 660.966,A -85,B 0,C 180,E1 -26486.683,E2 -26486.683} C_VEL
LIN {X 0,Y 124.236,Z 666.105,A -85,B 0,C 180,E1 -26491.945,E2 -26491.945} C_VEL
LIN {X 0,Y 115.902,Z 670.055,A -85,B 0,C 180,E1 -26497.974,E2 -26497.974} C_VEL
LIN {X 0,Y 108.358,Z 673.047,A -85,B 0,C 180,E1 -26505.519,E2 -26505.519} C_VEL
LIN {X 0,Y 103.599,Z 674.603,A -85,B 0,C 180,E1 -26512.37,E2 -26512.37} C_VEL
LIN {X 0,Y 99.952,Z 675.257,A -85,B 0,C 180,E1 -26520.514,E2 -26520.514} C_VEL
LIN {X 0,Y 98.071,Z 674.964,A -85,B 0,C 180,E1 -26529.003,E2 -26529.003} C_VEL
LIN {X 0,Y 97.46,Z 673.64,A -85,B 0,C 180,E1 -26537.506,E2 -26537.506} C_VEL
LIN {X 0,Y 98.521,Z 670.918,A -85,B 0,C 180,E1 -26547.118,E2 -26547.118} C_VEL
LIN {X 0,Y 100.493,Z 667.128,A -85,B 0,C 180,E1 -26556.021,E2 -26556.021} C_VEL
LIN {X 0,Y 103.874,Z 662.543,A -85,B 0,C 180,E1 -26563.698,E2 -26563.698} C_VEL
LIN {X 0,Y 108.656,Z 656.84,A -85,B 0,C 180,E1 -26570.839,E2 -26570.839} C_VEL
LIN {X 0,Y 115.825,Z 648.937,A -85,B 0,C 180,E1 -26578.05,E2 -26578.05} C_VEL
LIN {X 0,Y 123.43,Z 640.438,A -85,B 0,C 180,E1 -26583.721,E2 -26583.721} C_VEL
LIN {X 0,Y 131.957,Z 630.246,A -85,B 0,C 180,E1 -26588.741,E2 -26588.741} C_VEL
LIN {X 0,Y 140.117,Z 619.715,A -85,B 0,C 180,E1 -26592.62,E2 -26592.62} C_VEL
LIN {X 0,Y 148.674,Z 607.399,A -85,B 0,C 180,E1 -26596.127,E2 -26596.127} C_VEL
LIN {X 0,Y 156.387,Z 595.021,A -85,B 0,C 180,E1 -26598.828,E2 -26598.828} C_VEL
LIN {X 0,Y 163.761,Z 581.603,A -85,B 0,C 180,E1 -26601.065,E2 -26601.065} C_VEL
LIN {X 0,Y 170.558,Z 567.055,A -85,B 0,C 180,E1 -26602.974,E2 -26602.974} C_VEL
LIN {X 0,Y 176.092,Z 553.087,A -85,B 0,C 180,E1 -26604.408,E2 -26604.408} C_VEL
LIN {X 0,Y 181.093,Z 538.151,A -85,B 0,C 180,E1 -26605.557,E2 -26605.557} C_VEL
LIN {X 0,Y 185.559,Z 520.785,A -85,B 0,C 180,E1 -26606.556,E2 -26606.556} C_VEL
LIN {X 0,Y 188.65,Z 503.991,A -85,B 0,C 180,E1 -26607.196,E2 -26607.196} C_VEL
LIN {X 0,Y 191.845,Z 474.754,A -85,B 0,C 180,E1 -26607.949,E2 -26607.949} C_VEL
LIN {X 0,Y 195.914,Z 433.41,A -85,B 0,C 180,E1 -26608.977,E2 -26608.977} C_VEL
LIN {X 0,Y 192.376,Z 425.224,A -85,B 0,C 180,E1 -26612.334,E2 -26612.334} C_VEL
LIN {X 0,Y 189.509,Z 418.96,A -85,B 0,C 180,E1 -26615.571,E2 -26615.571} C_VEL
LIN {X 0,Y 187.158,Z 414.21,A -85,B 0,C 180,E1 -26618.775,E2 -26618.775} C_VEL
LIN {X 0,Y 185.209,Z 410.501,A -85,B 0,C 180,E1 -26622.099,E2 -26622.099} C_VEL
LIN {X 0,Y 183.524,Z 407.018,A -85,B 0,C 180,E1 -26626.286,E2 -26626.286} C_VEL
LIN {X 0,Y 182.463,Z 405.062,A -85,B 0,C 180,E1 -26632.349,E2 -26632.349} C_VEL
LIN {X 0,Y 182.566,Z 405.12,A -85,B 0,C 180,E1 -26635.583,E2 -26635.583} C_VEL
LIN {X 0,Y 183.127,Z 406.074,A -85,B 0,C 180,E1 -26638.83,E2 -26638.83} C_VEL
LIN {X 0,Y 183.879,Z 407.252,A -85,B 0,C 180,E1 -26641.262,E2 -26641.262} C_VEL
LIN {X 0,Y 185.773,Z 411.349,A -85,B 0,C 180,E1 -26645.528,E2 -26645.528} C_VEL
LIN {X 0,Y 187.679,Z 415.262,A -85,B 0,C 180,E1 -26648.613,E2 -26648.613} C_VEL
LIN {X 0,Y 190.339,Z 420.642,A -85,B 0,C 180,E1 -26652.028,E2 -26652.028} C_VEL
LIN {X 0,Y 193.564,Z 427.817,A -85,B 0,C 180,E1 -26655.457,E2 -26655.457} C_VEL
LIN {X 0,Y 196.044,Z 433.637,A -85,B 0,C 180,E1 -26657.738,E2 -26657.738} C_VEL
LIN {X 0,Y 188.635,Z 506.702,A -85,B 0,C 180,E1 -26659.556,E2 -26659.556} C_VEL
LIN {X 0,Y 185.754,Z 522.971,A -85,B 0,C 180,E1 -26660.153,E2 -26660.153} C_VEL
LIN {X 0,Y 181.581,Z 539.546,A -85,B 0,C 180,E1 -26660.974,E2 -26660.974} C_VEL
LIN {X 0,Y 176.298,Z 555.644,A -85,B 0,C 180,E1 -26662.052,E2 -26662.052} C_VEL
LIN {X 0,Y 170.492,Z 570.531,A -85,B 0,C 180,E1 -26663.482,E2 -26663.482} C_VEL
LIN {X 0,Y 163.214,Z 585.728,A -85,B 0,C 180,E1 -26665.277,E2 -26665.277} C_VEL
LIN {X 0,Y 155.549,Z 599.641,A -85,B 0,C 180,E1 -26667.54,E2 -26667.54} C_VEL
LIN {X 0,Y 148.096,Z 611.469,A -85,B 0,C 180,E1 -26669.996,E2 -26669.996} C_VEL
LIN {X 0,Y 140.289,Z 622.8,A -85,B 0,C 180,E1 -26673.044,E2 -26673.044} C_VEL
LIN {X 0,Y 131.852,Z 633.832,A -85,B 0,C 180,E1 -26676.915,E2 -26676.915} C_VEL
LIN {X 0,Y 122.945,Z 644.559,A -85,B 0,C 180,E1 -26682.002,E2 -26682.002} C_VEL
LIN {X 0,Y 115.157,Z 653.558,A -85,B 0,C 180,E1 -26687.86,E2 -26687.86} C_VEL
LIN {X 0,Y 108.657,Z 661.008,A -85,B 0,C 180,E1 -26694.4,E2 -26694.4} C_VEL
LIN {X 0,Y 103.88,Z 666.792,A -85,B 0,C 180,E1 -26701.162,E2 -26701.162} C_VEL
LIN {X 0,Y 101.678,Z 668.916,A -85,B 0,C 180,E1 -26703.981,E2 -26703.981} C_VEL
LIN {X 0,Y 96.814,Z 671.94,A -85,B 0,C 180,E1 -26708.66,E2 -26708.66} C_VEL
LIN {X 0,Y 93.186,Z 673.968,A -85,B 0,C 180,E1 -26712.772,E2 -26712.772} C_VEL
LIN {X 0,Y 91.476,Z 675.308,A -85,B 0,C 180,E1 -26716.208,E2 -26716.208} C_VEL
LIN {X 0,Y 91.221,Z 675.723,A -85,B 0,C 180,E1 -26717.413,E2 -26717.413} C_VEL
LIN {X 0,Y 90.863,Z 678.164,A -85,B 0,C 180,E1 -26725.564,E2 -26725.564} C_VEL
LIN {X 0,Y 91.036,Z 679.14,A -85,B 0,C 180,E1 -26730.001,E2 -26730.001} C_VEL
LIN {X 0,Y 90.921,Z 680.295,A -85,B 0,C 180,E1 -26738.894,E2 -26738.894} C_VEL
LIN {X 0,Y 92.253,Z 680.461,A -85,B 0,C 180,E1 -26747.742,E2 -26747.742} C_VEL
LIN {X 0,Y 95.475,Z 679.719,A -85,B 0,C 180,E1 -26756.211,E2 -26756.211} C_VEL
LIN {X 0,Y 100.494,Z 678.045,A -85,B 0,C 180,E1 -26764.02,E2 -26764.02} C_VEL
LIN {X 0,Y 107.118,Z 675.421,A -85,B 0,C 180,E1 -26771.003,E2 -26771.003} C_VEL
LIN {X 0,Y 115.082,Z 671.829,A -85,B 0,C 180,E1 -26777.125,E2 -26777.125} C_VEL
LIN {X 0,Y 124.247,Z 667.197,A -85,B 0,C 180,E1 -26782.365,E2 -26782.365} C_VEL
LIN {X 0,Y 134.306,Z 661.452,A -85,B 0,C 180,E1 -26786.852,E2 -26786.852} C_VEL
LIN {X 0,Y 145.101,Z 654.558,A -85,B 0,C 180,E1 -26790.673,E2 -26790.673} C_VEL
LIN {X 0,Y 156.461,Z 646.222,A -85,B 0,C 180,E1 -26793.945,E2 -26793.945} C_VEL
LIN {X 0,Y 168.313,Z 636.366,A -85,B 0,C 180,E1 -26796.726,E2 -26796.726} C_VEL
LIN {X 0,Y 179.013,Z 626.276,A -85,B 0,C 180,E1 -26798.816,E2 -26798.816} C_VEL
LIN {X 0,Y 189.881,Z 614.468,A -85,B 0,C 180,E1 -26800.705,E2 -26800.705} C_VEL
LIN {X 0,Y 200.221,Z 601.512,A -85,B 0,C 180,E1 -26802.199,E2 -26802.199} C_VEL
LIN {X 0,Y 208.285,Z 589.915,A -85,B 0,C 180,E1 -26803.224,E2 -26803.224} C_VEL
LIN {X 0,Y 216.368,Z 576.457,A -85,B 0,C 180,E1 -26804.212,E2 -26804.212} C_VEL
LIN {X 0,Y 224.558,Z 560.086,A -85,B 0,C 180,E1 -26805.083,E2 -26805.083} C_VEL
LIN {X 0,Y 230.743,Z 544.783,A -85,B 0,C 180,E1 -26805.686,E2 -26805.686} C_VEL
LIN {X 0,Y 235.954,Z 528.421,A -85,B 0,C 180,E1 -26806.176,E2 -26806.176} C_VEL
LIN {X 0,Y 239.857,Z 511.822,A -85,B 0,C 180,E1 -26806.525,E2 -26806.525} C_VEL
LIN {X 0,Y 242.35,Z 495.709,A -85,B 0,C 180,E1 -26806.841,E2 -26806.841} C_VEL
LIN {X 0,Y 244.471,Z 477.413,A -85,B 0,C 180,E1 -26807.171,E2 -26807.171} C_VEL
LIN {X 0,Y 243.718,Z 475.058,A -85,B 0,C 180,E1 -26809.766,E2 -26809.766} C_VEL
LIN {X 0,Y 243.276,Z 473.643,A -85,B 0,C 180,E1 -26813.365,E2 -26813.365} C_VEL
LIN {X 0,Y 243.631,Z 474.448,A -85,B 0,C 180,E1 -26817.107,E2 -26817.107} C_VEL
LIN {X 0,Y 243.971,Z 475.414,A -85,B 0,C 180,E1 -26818.557,E2 -26818.557} C_VEL
LIN {X 0,Y 244.493,Z 477.081,A -85,B 0,C 180,E1 -26820.232,E2 -26820.232} C_VEL
LIN {X 0,Y 241.046,Z 504.585,A -85,B 0,C 180,E1 -26820.737,E2 -26820.737} C_VEL
LIN {X 0,Y 237.458,Z 521.762,A -85,B 0,C 180,E1 -26821.076,E2 -26821.076} C_VEL
LIN {X 0,Y 233.328,Z 536.046,A -85,B 0,C 180,E1 -26821.549,E2 -26821.549} C_VEL
LIN {X 0,Y 227.473,Z 551.994,A -85,B 0,C 180,E1 -26822.229,E2 -26822.229} C_VEL
LIN {X 0,Y 221.673,Z 564.941,A -85,B 0,C 180,E1 -26822.928,E2 -26822.928} C_VEL
LIN {X 0,Y 213.961,Z 579.239,A -85,B 0,C 180,E1 -26823.897,E2 -26823.897} C_VEL
LIN {X 0,Y 205.489,Z 592.572,A -85,B 0,C 180,E1 -26825.049,E2 -26825.049} C_VEL
LIN {X 0,Y 196.265,Z 605.092,A -85,B 0,C 180,E1 -26826.436,E2 -26826.436} C_VEL
LIN {X 0,Y 186.341,Z 616.705,A -85,B 0,C 180,E1 -26828.092,E2 -26828.092} C_VEL
LIN {X 0,Y 174.992,Z 628.238,A -85,B 0,C 180,E1 -26830.272,E2 -26830.272} C_VEL
LIN {X 0,Y 163.926,Z 638.025,A -85,B 0,C 180,E1 -26832.743,E2 -26832.743} C_VEL
LIN {X 0,Y 153.225,Z 646.399,A -85,B 0,C 180,E1 -26835.589,E2 -26835.589} C_VEL
LIN {X 0,Y 141.485,Z 654.323,A -85,B 0,C 180,E1 -26839.301,E2 -26839.301} C_VEL
LIN {X 0,Y 130.484,Z 660.816,A -85,B 0,C 180,E1 -26843.703,E2 -26843.703} C_VEL
LIN {X 0,Y 120.393,Z 666.048,A -85,B 0,C 180,E1 -26848.879,E2 -26848.879} C_VEL
LIN {X 0,Y 111.392,Z 670.043,A -85,B 0,C 180,E1 -26854.894,E2 -26854.894} C_VEL
LIN {X 0,Y 102.428,Z 673.347,A -85,B 0,C 180,E1 -26863.328,E2 -26863.328} C_VEL
LIN {X 0,Y 97.716,Z 674.736,A -85,B 0,C 180,E1 -26869.66,E2 -26869.66} C_VEL
LIN {X 0,Y 93.499,Z 675.455,A -85,B 0,C 180,E1 -26878.252,E2 -26878.252} C_VEL
LIN {X 0,Y 91.105,Z 675.191,A -85,B 0,C 180,E1 -26887.78,E2 -26887.78} C_VEL
LIN {X 0,Y 90.353,Z 673.956,A -85,B 0,C 180,E1 -26896.505,E2 -26896.505} C_VEL
LIN {X 0,Y 91.069,Z 671.757,A -85,B 0,C 180,E1 -26905.573,E2 -26905.573} C_VEL
LIN {X 0,Y 91.828,Z 670.28,A -85,B 0,C 180,E1 -26909.999,E2 -26909.999} C_VEL
LIN {X 0,Y 95.054,Z 665.47,A -85,B 0,C 180,E1 -26920.651,E2 -26920.651} C_VEL
LIN {X 0,Y 99.295,Z 660.398,A -85,B 0,C 180,E1 -26928.572,E2 -26928.572} C_VEL
LIN {X 0,Y 105.208,Z 654.207,A -85,B 0,C 180,E1 -26935.734,E2 -26935.734} C_VEL
LIN {X 0,Y 113.457,Z 645.631,A -85,B 0,C 180,E1 -26942.82,E2 -26942.82} C_VEL
LIN {X 0,Y 121.939,Z 636.371,A -85,B 0,C 180,E1 -26948.285,E2 -26948.285} C_VEL
LIN {X 0,Y 130.119,Z 626.84,A -85,B 0,C 180,E1 -26952.466,E2 -26952.466} C_VEL
LIN {X 0,Y 138.741,Z 615.768,A -85,B 0,C 180,E1 -26956.206,E2 -26956.206} C_VEL
LIN {X 0,Y 146.515,Z 604.681,A -85,B 0,C 180,E1 -26959.068,E2 -26959.068} C_VEL
LIN {X 0,Y 153.876,Z 592.877,A -85,B 0,C 180,E1 -26961.458,E2 -26961.458} C_VEL
LIN {X 0,Y 161.523,Z 579.055,A -85,B 0,C 180,E1 -26963.605,E2 -26963.605} C_VEL
LIN {X 0,Y 168.536,Z 564.041,A -85,B 0,C 180,E1 -26965.444,E2 -26965.444} C_VEL
LIN {X 0,Y 174.993,Z 547.318,A -85,B 0,C 180,E1 -26966.969,E2 -26966.969} C_VEL
LIN {X 0,Y 180.126,Z 530.609,A -85,B 0,C 180,E1 -26968.062,E2 -26968.062} C_VEL
LIN {X 0,Y 184.008,Z 513.718,A -85,B 0,C 180,E1 -26968.846,E2 -26968.846} C_VEL
LIN {X 0,Y 186.628,Z 497.167,A -85,B 0,C 180,E1 -26969.344,E2 -26969.344} C_VEL
LIN {X 0,Y 192.76,Z 436.98,A -85,B 0,C 180,E1 -26970.84,E2 -26970.84} C_VEL
LIN {X 0,Y 189.542,Z 429.23,A -85,B 0,C 180,E1 -26974.285,E2 -26974.285} C_VEL
LIN {X 0,Y 187.089,Z 423.548,A -85,B 0,C 180,E1 -26977.467,E2 -26977.467} C_VEL
LIN {X 0,Y 184.928,Z 419.263,A -85,B 0,C 180,E1 -26980.848,E2 -26980.848} C_VEL
LIN {X 0,Y 183.829,Z 416.991,A -85,B 0,C 180,E1 -26983.026,E2 -26983.026} C_VEL
LIN {X 0,Y 182.519,Z 413.976,A -85,B 0,C 180,E1 -26986.641,E2 -26986.641} C_VEL
LIN {X 0,Y 181.58,Z 411.957,A -85,B 0,C 180,E1 -26993.331,E2 -26993.331} C_VEL
LIN {X 0,Y 182.02,Z 412.678,A -85,B 0,C 180,E1 -26997.786,E2 -26997.786} C_VEL
LIN {X 0,Y 182.823,Z 414.149,A -85,B 0,C 180,E1 -27000.815,E2 -27000.815} C_VEL
LIN {X 0,Y 184.45,Z 417.918,A -85,B 0,C 180,E1 -27004.797,E2 -27004.797} C_VEL
LIN {X 0,Y 186.256,Z 421.865,A -85,B 0,C 180,E1 -27007.938,E2 -27007.938} C_VEL
LIN {X 0,Y 188.561,Z 426.815,A -85,B 0,C 180,E1 -27011.113,E2 -27011.113} C_VEL
LIN {X 0,Y 191.405,Z 433.539,A -85,B 0,C 180,E1 -27014.383,E2 -27014.383} C_VEL
LIN {X 0,Y 192.889,Z 437.16,A -85,B 0,C 180,E1 -27015.883,E2 -27015.883} C_VEL
LIN {X 0,Y 185.688,Z 506.411,A -85,B 0,C 180,E1 -27017.575,E2 -27017.575} C_VEL
LIN {X 0,Y 182.813,Z 522.408,A -85,B 0,C 180,E1 -27018.144,E2 -27018.144} C_VEL
LIN {X 0,Y 178.746,Z 538.431,A -85,B 0,C 180,E1 -27018.899,E2 -27018.899} C_VEL
LIN {X 0,Y 173.349,Z 554.748,A -85,B 0,C 180,E1 -27019.936,E2 -27019.936} C_VEL
LIN {X 0,Y 167.715,Z 568.918,A -85,B 0,C 180,E1 -27021.193,E2 -27021.193} C_VEL
LIN {X 0,Y 161.01,Z 582.862,A -85,B 0,C 180,E1 -27022.766,E2 -27022.766} C_VEL
LIN {X 0,Y 153.725,Z 596.002,A -85,B 0,C 180,E1 -27024.682,E2 -27024.682} C_VEL
LIN {X 0,Y 145.977,Z 608.414,A -85,B 0,C 180,E1 -27027.042,E2 -27027.042} C_VEL
LIN {X 0,Y 136.549,Z 621.763,A -85,B 0,C 180,E1 -27030.449,E2 -27030.449} C_VEL
LIN {X 0,Y 127.613,Z 632.981,A -85,B 0,C 180,E1 -27034.301,E2 -27034.301} C_VEL
LIN {X 0,Y 119.369,Z 642.569,A -85,B 0,C 180,E1 -27038.73,E2 -27038.73} C_VEL
LIN {X 0,Y 111.275,Z 651.423,A -85,B 0,C 180,E1 -27044.174,E2 -27044.174} C_VEL
LIN {X 0,Y 104.508,Z 658.716,A -85,B 0,C 180,E1 -27050.294,E2 -27050.294} C_VEL
LIN {X 0,Y 98.552,Z 665.211,A -85,B 0,C 180,E1 -27057.667,E2 -27057.667} C_VEL
LIN {X 0,Y 94.286,Z 670.512,A -85,B 0,C 180,E1 -27065.798,E2 -27065.798} C_VEL
LIN {X 0,Y 92.157,Z 673.663,A -85,B 0,C 180,E1 -27072.24,E2 -27072.24} C_VEL
LIN {X 0,Y 91.221,Z 675.723,A -85,B 0,C 180,E1 -27077.413,E2 -27077.413} C_VEL
LIN {X 0,Y 90.183,Z 676.922,A -85,B 0,C 180,E1 -27081.023,E2 -27081.023} C_VEL
LIN {X 0,Y 88.411,Z 677.884,A -85,B 0,C 180,E1 -27084.623,E2 -27084.623} C_VEL
LIN {X 0,Y 83.943,Z 679.616,A -85,B 0,C 180,E1 -27094.877,E2 -27094.877} C_VEL
LIN {X 0,Y 83.734,Z 679.852,A -85,B 0,C 180,E1 -27097.624,E2 -27097.624} C_VEL
LIN {X 0,Y 85.444,Z 680.268,A -85,B 0,C 180,E1 -27109.209,E2 -27109.209} C_VEL
LIN {X 0,Y 89.088,Z 679.56,A -85,B 0,C 180,E1 -27118.251,E2 -27118.251} C_VEL
LIN {X 0,Y 94.619,Z 677.954,A -85,B 0,C 180,E1 -27126.457,E2 -27126.457} C_VEL
LIN {X 0,Y 101.789,Z 675.366,A -85,B 0,C 180,E1 -27133.666,E2 -27133.666} C_VEL
LIN {X 0,Y 110.324,Z 671.846,A -85,B 0,C 180,E1 -27139.858,E2 -27139.858} C_VEL
LIN {X 0,Y 122.565,Z 665.974,A -85,B 0,C 180,E1 -27146.248,E2 -27146.248} C_VEL
LIN {X 0,Y 136.094,Z 658.336,A -85,B 0,C 180,E1 -27151.39,E2 -27151.39} C_VEL
LIN {X 0,Y 149.011,Z 649.78,A -85,B 0,C 180,E1 -27155.22,E2 -27155.22} C_VEL
LIN {X 0,Y 161.023,Z 640.591,A -85,B 0,C 180,E1 -27158.046,E2 -27158.046} C_VEL
LIN {X 0,Y 173.424,Z 629.729,A -85,B 0,C 180,E1 -27160.426,E2 -27160.426} C_VEL
LIN {X 0,Y 184.462,Z 618.568,A -85,B 0,C 180,E1 -27162.27,E2 -27162.27} C_VEL
LIN {X 0,Y 194.94,Z 606.466,A -85,B 0,C 180,E1 -27163.718,E2 -27163.718} C_VEL
LIN {X 0,Y 205.531,Z 592.099,A -85,B 0,C 180,E1 -27165.015,E2 -27165.015} C_VEL
LIN {X 0,Y 214.566,Z 577.507,A -85,B 0,C 180,E1 -27166.014,E2 -27166.014} C_VEL
LIN {X 0,Y 222.03,Z 563.166,A -85,B 0,C 180,E1 -27166.742,E2 -27166.742} C_VEL
LIN {X 0,Y 228.685,Z 547.675,A -85,B 0,C 180,E1 -27167.357,E2 -27167.357} C_VEL
LIN {X 0,Y 234.132,Z 531.79,A -85,B 0,C 180,E1 -27167.804,E2 -27167.804} C_VEL
LIN {X 0,Y 238.348,Z 515.345,A -85,B 0,C 180,E1 -27168.145,E2 -27168.145} C_VEL
LIN {X 0,Y 241.074,Z 499.428,A -85,B 0,C 180,E1 -27168.445,E2 -27168.445} C_VEL
LIN {X 0,Y 243.072,Z 483.136,A -85,B 0,C 180,E1 -27168.717,E2 -27168.717} C_VEL
LIN {X 0,Y 242.78,Z 482.032,A -85,B 0,C 180,E1 -27169.999,E2 -27169.999} C_VEL
LIN {X 0,Y 242.393,Z 480.695,A -85,B 0,C 180,E1 -27173.934,E2 -27173.934} C_VEL
LIN {X 0,Y 242.892,Z 481.788,A -85,B 0,C 180,E1 -27177.721,E2 -27177.721} C_VEL
LIN {X 0,Y 243.096,Z 482.728,A -85,B 0,C 180,E1 -27178.655,E2 -27178.655} C_VEL
LIN {X 0,Y 240.054,Z 505.78,A -85,B 0,C 180,E1 -27179.08,E2 -27179.08} C_VEL
LIN {X 0,Y 236.489,Z 522.456,A -85,B 0,C 180,E1 -27179.387,E2 -27179.387} C_VEL
LIN {X 0,Y 232.303,Z 536.62,A -85,B 0,C 180,E1 -27179.825,E2 -27179.825} C_VEL
LIN {X 0,Y 226.284,Z 552.679,A -85,B 0,C 180,E1 -27180.47,E2 -27180.47} C_VEL
LIN {X 0,Y 220.546,Z 565.267,A -85,B 0,C 180,E1 -27181.109,E2 -27181.109} C_VEL
LIN {X 0,Y 212.59,Z 579.76,A -85,B 0,C 180,E1 -27182.026,E2 -27182.026} C_VEL
LIN {X 0,Y 204.109,Z 592.857,A -85,B 0,C 180,E1 -27183.088,E2 -27183.088} C_VEL
LIN {X 0,Y 194.657,Z 605.439,A -85,B 0,C 180,E1 -27184.397,E2 -27184.397} C_VEL
LIN {X 0,Y 183.761,Z 617.879,A -85,B 0,C 180,E1 -27186.075,E2 -27186.075} C_VEL
LIN {X 0,Y 172.168,Z 629.234,A -85,B 0,C 180,E1 -27188.147,E2 -27188.147} C_VEL
LIN {X 0,Y 160.781,Z 638.916,A -85,B 0,C 180,E1 -27190.519,E2 -27190.519} C_VEL
LIN {X 0,Y 148.007,Z 648.356,A -85,B 0,C 180,E1 -27193.736,E2 -27193.736} C_VEL
LIN {X 0,Y 136.212,Z 655.88,A -85,B 0,C 180,E1 -27197.344,E2 -27197.344} C_VEL
LIN {X 0,Y 124.859,Z 662.124,A -85,B 0,C 180,E1 -27201.759,E2 -27201.759} C_VEL
LIN {X 0,Y 114.384,Z 667.077,A -85,B 0,C 180,E1 -27207.011,E2 -27207.011} C_VEL
LIN {X 0,Y 107.087,Z 670.089,A -85,B 0,C 180,E1 -27211.673,E2 -27211.673} C_VEL
LIN {X 0,Y 96.64,Z 673.652,A -85,B 0,C 180,E1 -27220.886,E2 -27220.886} C_VEL
LIN {X 0,Y 92.099,Z 674.853,A -85,B 0,C 180,E1 -27226.623,E2 -27226.623} C_VEL
LIN {X 0,Y 87.209,Z 675.653,A -85,B 0,C 180,E1 -27235.658,E2 -27235.658} C_VEL
LIN {X 0,Y 84.144,Z 675.374,A -85,B 0,C 180,E1 -27246.752,E2 -27246.752} C_VEL
LIN {X 0,Y 83.263,Z 674.269,A -85,B 0,C 180,E1 -27255.331,E2 -27255.331} C_VEL
LIN {X 0,Y 83.878,Z 672.145,A -85,B 0,C 180,E1 -27265.193,E2 -27265.193} C_VEL
LIN {X 0,Y 84.691,Z 670.666,A -85,B 0,C 180,E1 -27269.999,E2 -27269.999} C_VEL
LIN {X 0,Y 88.094,Z 665.936,A -85,B 0,C 180,E1 -27281.504,E2 -27281.504} C_VEL
LIN {X 0,Y 92.611,Z 660.951,A -85,B 0,C 180,E1 -27289.967,E2 -27289.967} C_VEL
LIN {X 0,Y 98.867,Z 654.838,A -85,B 0,C 180,E1 -27297.519,E2 -27297.519} C_VEL
LIN {X 0,Y 107.582,Z 646.331,A -85,B 0,C 180,E1 -27304.862,E2 -27304.862} C_VEL
LIN {X 0,Y 116.482,Z 637.174,A -85,B 0,C 180,E1 -27310.436,E2 -27310.436} C_VEL
LIN {X 0,Y 126.263,Z 626.291,A -85,B 0,C 180,E1 -27315.209,E2 -27315.209} C_VEL
LIN {X 0,Y 135.282,Z 615.069,A -85,B 0,C 180,E1 -27318.875,E2 -27318.875} C_VEL
LIN {X 0,Y 144.046,Z 602.873,A -85,B 0,C 180,E1 -27321.881,E2 -27321.881} C_VEL
LIN {X 0,Y 152.419,Z 589.567,A -85,B 0,C 180,E1 -27324.359,E2 -27324.359} C_VEL
LIN {X 0,Y 160.353,Z 574.986,A -85,B 0,C 180,E1 -27326.38,E2 -27326.38} C_VEL
LIN {X 0,Y 166.826,Z 560.728,A -85,B 0,C 180,E1 -27327.975,E2 -27327.975} C_VEL
LIN {X 0,Y 172.773,Z 545.232,A -85,B 0,C 180,E1 -27329.24,E2 -27329.24} C_VEL
LIN {X 0,Y 177.646,Z 529.345,A -85,B 0,C 180,E1 -27330.213,E2 -27330.213} C_VEL
LIN {X 0,Y 181.617,Z 512.007,A -85,B 0,C 180,E1 -27330.962,E2 -27330.962} C_VEL
LIN {X 0,Y 184.26,Z 494.409,A -85,B 0,C 180,E1 -27331.449,E2 -27331.449} C_VEL
LIN {X 0,Y 189.831,Z 441.1,A -85,B 0,C 180,E1 -27332.689,E2 -27332.689} C_VEL
LIN {X 0,Y 189.525,Z 439.883,A -85,B 0,C 180,E1 -27333.079,E2 -27333.079} C_VEL
LIN {X 0,Y 186.479,Z 432.167,A -85,B 0,C 180,E1 -27336.918,E2 -27336.918} C_VEL
LIN {X 0,Y 184.32,Z 427.285,A -85,B 0,C 180,E1 -27340.272,E2 -27340.272} C_VEL
LIN {X 0,Y 182.801,Z 423.988,A -85,B 0,C 180,E1 -27343.281,E2 -27343.281} C_VEL
LIN {X 0,Y 181.451,Z 420.858,A -85,B 0,C 180,E1 -27347.24,E2 -27347.24} C_VEL
LIN {X 0,Y 180.704,Z 419.01,A -85,B 0,C 180,E1 -27353.298,E2 -27353.298} C_VEL
LIN {X 0,Y 181.134,Z 419.762,A -85,B 0,C 180,E1 -27357.775,E2 -27357.775} C_VEL
LIN {X 0,Y 181.817,Z 421.187,A -85,B 0,C 180,E1 -27360.508,E2 -27360.508} C_VEL
LIN {X 0,Y 183.266,Z 424.766,A -85,B 0,C 180,E1 -27364.295,E2 -27364.295} C_VEL
LIN {X 0,Y 184.923,Z 428.626,A -85,B 0,C 180,E1 -27367.361,E2 -27367.361} C_VEL
LIN {X 0,Y 187.512,Z 434.622,A -85,B 0,C 180,E1 -27371.082,E2 -27371.082} C_VEL
LIN {X 0,Y 189.936,Z 440.923,A -85,B 0,C 180,E1 -27373.988,E2 -27373.988} C_VEL
LIN {X 0,Y 183.039,Z 505.716,A -85,B 0,C 180,E1 -27375.537,E2 -27375.537} C_VEL
LIN {X 0,Y 180.074,Z 521.987,A -85,B 0,C 180,E1 -27376.078,E2 -27376.078} C_VEL
LIN {X 0,Y 176.523,Z 536.063,A -85,B 0,C 180,E1 -27376.69,E2 -27376.69} C_VEL
LIN {X 0,Y 171.42,Z 551.808,A -85,B 0,C 180,E1 -27377.595,E2 -27377.595} C_VEL
LIN {X 0,Y 165.221,Z 567.18,A -85,B 0,C 180,E1 -27378.837,E2 -27378.837} C_VEL
LIN {X 0,Y 158.357,Z 581.425,A -85,B 0,C 180,E1 -27380.358,E2 -27380.358} C_VEL
LIN {X 0,Y 150.108,Z 595.979,A -85,B 0,C 180,E1 -27382.379,E2 -27382.379} C_VEL
LIN {X 0,Y 142.115,Z 608.361,A -85,B 0,C 180,E1 -27384.674,E2 -27384.674} C_VEL
LIN {X 0,Y 133.017,Z 620.788,A -85,B 0,C 180,E1 -27387.75,E2 -27387.75} C_VEL
LIN {X 0,Y 123.671,Z 632.128,A -85,B 0,C 180,E1 -27391.524,E2 -27391.524} C_VEL
LIN {X 0,Y 114.97,Z 641.826,A -85,B 0,C 180,E1 -27395.909,E2 -27395.909} C_VEL
LIN {X 0,Y 106.352,Z 650.767,A -85,B 0,C 180,E1 -27401.36,E2 -27401.36} C_VEL
LIN {X 0,Y 99.036,Z 658.115,A -85,B 0,C 180,E1 -27407.612,E2 -27407.612} C_VEL
LIN {X 0,Y 92.515,Z 664.694,A -85,B 0,C 180,E1 -27415.268,E2 -27415.268} C_VEL
LIN {X 0,Y 87.758,Z 670.069,A -85,B 0,C 180,E1 -27423.867,E2 -27423.867} C_VEL
LIN {X 0,Y 84.359,Z 675.092,A -85,B 0,C 180,E1 -27435.527,E2 -27435.527} C_VEL
LIN {X 0,Y 83.764,Z 677.84,A -85,B 0,C 180,E1 -27445.188,E2 -27445.188} C_VEL
LIN {X 0,Y 83.932,Z 678.85,A -85,B 0,C 180,E1 -27450.001,E2 -27450.001} C_VEL
LIN {X 0,Y 83.734,Z 679.852,A -85,B 0,C 180,E1 -27457.624,E2 -27457.624} C_VEL
LIN {X 0,Y 83.372,Z 680.165,A -85,B 0,C 180,E1 -27461.656,E2 -27461.656} C_VEL
LIN {X 0,Y 81.699,Z 680.214,A -85,B 0,C 180,E1 -27468.442,E2 -27468.442} C_VEL
LIN {X 0,Y 80.958,Z 679.963,A -85,B 0,C 180,E1 -27474.042,E2 -27474.042} C_VEL
LIN {X 0,Y 81.661,Z 679.67,A -85,B 0,C 180,E1 -27478.195,E2 -27478.195} C_VEL
LIN {X 0,Y 82.243,Z 679.51,A -85,B 0,C 180,E1 -27479.515,E2 -27479.515} C_VEL
LIN {X 0,Y 88.943,Z 677.864,A -85,B 0,C 180,E1 -27489.208,E2 -27489.208} C_VEL
LIN {X 0,Y 96.706,Z 675.31,A -85,B 0,C 180,E1 -27496.615,E2 -27496.615} C_VEL
LIN {X 0,Y 108.605,Z 670.657,A -85,B 0,C 180,E1 -27504.383,E2 -27504.383} C_VEL
LIN {X 0,Y 121.452,Z 664.644,A -85,B 0,C 180,E1 -27510.227,E2 -27510.227} C_VEL
LIN {X 0,Y 132.815,Z 658.497,A -85,B 0,C 180,E1 -27514.102,E2 -27514.102} C_VEL
LIN {X 0,Y 146.165,Z 650.005,A -85,B 0,C 180,E1 -27517.758,E2 -27517.758} C_VEL
LIN {X 0,Y 158.503,Z 640.926,A -85,B 0,C 180,E1 -27520.429,E2 -27520.429} C_VEL
LIN {X 0,Y 171.178,Z 630.181,A -85,B 0,C 180,E1 -27522.664,E2 -27522.664} C_VEL
LIN {X 0,Y 182.437,Z 619.149,A -85,B 0,C 180,E1 -27524.383,E2 -27524.383} C_VEL
LIN {X 0,Y 192.266,Z 608.106,A -85,B 0,C 180,E1 -27525.621,E2 -27525.621} C_VEL
LIN {X 0,Y 202.155,Z 595.251,A -85,B 0,C 180,E1 -27526.764,E2 -27526.764} C_VEL
LIN {X 0,Y 211.32,Z 581.361,A -85,B 0,C 180,E1 -27527.674,E2 -27527.674} C_VEL
LIN {X 0,Y 218.852,Z 567.934,A -85,B 0,C 180,E1 -27528.365,E2 -27528.365} C_VEL
LIN {X 0,Y 225.577,Z 553.461,A -85,B 0,C 180,E1 -27528.934,E2 -27528.934} C_VEL
LIN {X 0,Y 231.501,Z 537.803,A -85,B 0,C 180,E1 -27529.399,E2 -27529.399} C_VEL
LIN {X 0,Y 236.197,Z 521.797,A -85,B 0,C 180,E1 -27529.732,E2 -27529.732} C_VEL
LIN {X 0,Y 239.668,Z 505.185,A -85,B 0,C 180,E1 -27530.045,E2 -27530.045} C_VEL
LIN {X 0,Y 241.832,Z 488.944,A -85,B 0,C 180,E1 -27530.318,E2 -27530.318} C_VEL
LIN {X 0,Y 241.52,Z 487.791,A -85,B 0,C 180,E1 -27533.317,E2 -27533.317} C_VEL
LIN {X 0,Y 241.785,Z 488.405,A -85,B 0,C 180,E1 -27536.668,E2 -27536.668} C_VEL
LIN {X 0,Y 241.858,Z 488.57,A -85,B 0,C 180,E1 -27537.05,E2 -27537.05} C_VEL
LIN {X 0,Y 239.199,Z 507.297,A -85,B 0,C 180,E1 -27537.401,E2 -27537.401} C_VEL
LIN {X 0,Y 235.528,Z 523.818,A -85,B 0,C 180,E1 -27537.698,E2 -27537.698} C_VEL
LIN {X 0,Y 231.212,Z 538.043,A -85,B 0,C 180,E1 -27538.121,E2 -27538.121} C_VEL
LIN {X 0,Y 225.533,Z 552.849,A -85,B 0,C 180,E1 -27538.677,E2 -27538.677} C_VEL
LIN {X 0,Y 219.644,Z 565.594,A -85,B 0,C 180,E1 -27539.274,E2 -27539.274} C_VEL
LIN {X 0,Y 211.452,Z 580.276,A -85,B 0,C 180,E1 -27540.134,E2 -27540.134} C_VEL
LIN {X 0,Y 202.972,Z 593.141,A -85,B 0,C 180,E1 -27541.102,E2 -27541.102} C_VEL
LIN {X 0,Y 194.253,Z 604.661,A -85,B 0,C 180,E1 -27542.217,E2 -27542.217} C_VEL
LIN {X 0,Y 184.828,Z 615.376,A -85,B 0,C 180,E1 -27543.485,E2 -27543.485} C_VEL
LIN {X 0,Y 172.944,Z 627.184,A -85,B 0,C 180,E1 -27545.361,E2 -27545.361} C_VEL
LIN {X 0,Y 161.502,Z 637.049,A -85,B 0,C 180,E1 -27547.503,E2 -27547.503} C_VEL
LIN {X 0,Y 149.873,Z 645.698,A -85,B 0,C 180,E1 -27550.015,E2 -27550.015} C_VEL
LIN {X 0,Y 137.231,Z 653.823,A -85,B 0,C 180,E1 -27553.332,E2 -27553.332} C_VEL
LIN {X 0,Y 125.151,Z 660.514,A -85,B 0,C 180,E1 -27557.319,E2 -27557.319} C_VEL
LIN {X 0,Y 113.833,Z 665.914,A -85,B 0,C 180,E1 -27562.165,E2 -27562.165} C_VEL
LIN {X 0,Y 102.392,Z 670.423,A -85,B 0,C 180,E1 -27568.719,E2 -27568.719} C_VEL
LIN {X 0,Y 91.08,Z 673.951,A -85,B 0,C 180,E1 -27578.123,E2 -27578.123} C_VEL
LIN {X 0,Y 83.672,Z 675.529,A -85,B 0,C 180,E1 -27587.781,E2 -27587.781} C_VEL
LIN {X 0,Y 79.089,Z 675.941,A -85,B 0,C 180,E1 -27597.779,E2 -27597.779} C_VEL
LIN {X 0,Y 76.729,Z 675.269,A -85,B 0,C 180,E1 -27608.507,E2 -27608.507} C_VEL
LIN {X 0,Y 76.199,Z 673.673,A -85,B 0,C 180,E1 -27619.369,E2 -27619.369} C_VEL
LIN {X 0,Y 77.555,Z 671.052,A -85,B 0,C 180,E1 -27629.999,E2 -27629.999} C_VEL
LIN {X 0,Y 81.155,Z 666.403,A -85,B 0,C 180,E1 -27642.503,E2 -27642.503} C_VEL
LIN {X 0,Y 85.994,Z 661.503,A -85,B 0,C 180,E1 -27651.578,E2 -27651.578} C_VEL
LIN {X 0,Y 92.639,Z 655.438,A -85,B 0,C 180,E1 -27659.545,E2 -27659.545} C_VEL
LIN {X 0,Y 101.862,Z 647.026,A -85,B 0,C 180,E1 -27667.135,E2 -27667.135} C_VEL
LIN {X 0,Y 111.207,Z 637.977,A -85,B 0,C 180,E1 -27672.794,E2 -27672.794} C_VEL
LIN {X 0,Y 121.381,Z 627.22,A -85,B 0,C 180,E1 -27677.58,E2 -27677.58} C_VEL
LIN {X 0,Y 130.767,Z 616.135,A -85,B 0,C 180,E1 -27681.195,E2 -27681.195} C_VEL
LIN {X 0,Y 139.113,Z 605.047,A -85,B 0,C 180,E1 -27683.932,E2 -27683.932} C_VEL
LIN {X 0,Y 147.71,Z 592.068,A -85,B 0,C 180,E1 -27686.371,E2 -27686.371} C_VEL
LIN {X 0,Y 155.82,Z 577.986,A -85,B 0,C 180,E1 -27688.356,E2 -27688.356} C_VEL
LIN {X 0,Y 162.48,Z 564.373,A -85,B 0,C 180,E1 -27689.892,E2 -27689.892} C_VEL
LIN {X 0,Y 169.286,Z 547.618,A -85,B 0,C 180,E1 -27691.284,E2 -27691.284} C_VEL
LIN {X 0,Y 174.652,Z 530.896,A -85,B 0,C 180,E1 -27692.286,E2 -27692.286} C_VEL
LIN {X 0,Y 178.702,Z 513.964,A -85,B 0,C 180,E1 -27693.002,E2 -27693.002} C_VEL
LIN {X 0,Y 181.395,Z 497.601,A -85,B 0,C 180,E1 -27693.445,E2 -27693.445} C_VEL
LIN {X 0,Y 187.095,Z 444.552,A -85,B 0,C 180,E1 -27694.688,E2 -27694.688} C_VEL
LIN {X 0,Y 184.659,Z 437.949,A -85,B 0,C 180,E1 -27698.122,E2 -27698.122} C_VEL
LIN {X 0,Y 182.711,Z 433.317,A -85,B 0,C 180,E1 -27701.482,E2 -27701.482} C_VEL
LIN {X 0,Y 181.471,Z 430.429,A -85,B 0,C 180,E1 -27704.269,E2 -27704.269} C_VEL
LIN {X 0,Y 180.493,Z 427.822,A -85,B 0,C 180,E1 -27707.513,E2 -27707.513} C_VEL
LIN {X 0,Y 179.828,Z 426.056,A -85,B 0,C 180,E1 -27713.266,E2 -27713.266} C_VEL
LIN {X 0,Y 180.169,Z 426.679,A -85,B 0,C 180,E1 -27717.322,E2 -27717.322} C_VEL
LIN {X 0,Y 180.811,Z 428.185,A -85,B 0,C 180,E1 -27720.17,E2 -27720.17} C_VEL
LIN {X 0,Y 182.133,Z 431.717,A -85,B 0,C 180,E1 -27723.871,E2 -27723.871} C_VEL
LIN {X 0,Y 183.711,Z 435.647,A -85,B 0,C 180,E1 -27726.953,E2 -27726.953} C_VEL
LIN {X 0,Y 185.833,Z 440.909,A -85,B 0,C 180,E1 -27730.21,E2 -27730.21} C_VEL
LIN {X 0,Y 187.205,Z 444.866,A -85,B 0,C 180,E1 -27732.064,E2 -27732.064} C_VEL
LIN {X 0,Y 180.419,Z 506.473,A -85,B 0,C 180,E1 -27733.463,E2 -27733.463} C_VEL
LIN {X 0,Y 177.185,Z 523.315,A -85,B 0,C 180,E1 -27734.001,E2 -27734.001} C_VEL
LIN {X 0,Y 173.003,Z 538.835,A -85,B 0,C 180,E1 -27734.682,E2 -27734.682} C_VEL
LIN {X 0,Y 167.38,Z 554.959,A -85,B 0,C 180,E1 -27735.613,E2 -27735.613} C_VEL
LIN {X 0,Y 161.473,Z 569.023,A -85,B 0,C 180,E1 -27736.758,E2 -27736.758} C_VEL
LIN {X 0,Y 153.703,Z 584.268,A -85,B 0,C 180,E1 -27738.358,E2 -27738.358} C_VEL
LIN {X 0,Y 145.998,Z 597.162,A -85,B 0,C 180,E1 -27740.169,E2 -27740.169} C_VEL
LIN {X 0,Y 138.509,Z 608.308,A -85,B 0,C 180,E1 -27742.18,E2 -27742.18} C_VEL
LIN {X 0,Y 129.809,Z 619.81,A -85,B 0,C 180,E1 -27744.926,E2 -27744.926} C_VEL
LIN {X 0,Y 120.054,Z 631.279,A -85,B 0,C 180,E1 -27748.586,E2 -27748.586} C_VEL
LIN {X 0,Y 110.872,Z 641.083,A -85,B 0,C 180,E1 -27752.871,E2 -27752.871} C_VEL
LIN {X 0,Y 101.03,Z 650.734,A -85,B 0,C 180,E1 -27758.758,E2 -27758.758} C_VEL
LIN {X 0,Y 91.865,Z 659.348,A -85,B 0,C 180,E1 -27766.486,E2 -27766.486} C_VEL
LIN {X 0,Y 85.164,Z 665.639,A -85,B 0,C 180,E1 -27774.714,E2 -27774.714} C_VEL
LIN {X 0,Y 80.323,Z 670.731,A -85,B 0,C 180,E1 -27784.057,E2 -27784.057} C_VEL
LIN {X 0,Y 77.44,Z 674.693,A -85,B 0,C 180,E1 -27794.202,E2 -27794.202} C_VEL
LIN {X 0,Y 76.649,Z 677.513,A -85,B 0,C 180,E1 -27804.74,E2 -27804.74} C_VEL
LIN {X 0,Y 76.836,Z 678.558,A -85,B 0,C 180,E1 -27810.001,E2 -27810.001} C_VEL
LIN {X 0,Y 76.839,Z 679.776,A -85,B 0,C 180,E1 -27820.541,E2 -27820.541} C_VEL
LIN {X 0,Y 78.701,Z 680.076,A -85,B 0,C 180,E1 -27830.929,E2 -27830.929} C_VEL
LIN {X 0,Y 82.243,Z 679.51,A -85,B 0,C 180,E1 -27839.515,E2 -27839.515} C_VEL
LIN {X 0,Y 83.821,Z 679.078,A -85,B 0,C 180,E1 -27843.428,E2 -27843.428} C_VEL
LIN {X 0,Y 85.545,Z 677.98,A -85,B 0,C 180,E1 -27849.994,E2 -27849.994} C_VEL
LIN {X 0,Y 87.539,Z 676.847,A -85,B 0,C 180,E1 -27855.038,E2 -27855.038} C_VEL
LIN {X 0,Y 90.132,Z 675.86,A -85,B 0,C 180,E1 -27858.409,E2 -27858.409} C_VEL
LIN {X 0,Y 91.28,Z 675.444,A -85,B 0,C 180,E1 -27859.397,E2 -27859.397} C_VEL
LIN {X 0,Y 101.66,Z 671.867,A -85,B 0,C 180,E1 -27866.058,E2 -27866.058} C_VEL
LIN {X 0,Y 115.201,Z 666.115,A -85,B 0,C 180,E1 -27872.202,E2 -27872.202} C_VEL
LIN {X 0,Y 126.86,Z 660.251,A -85,B 0,C 180,E1 -27876.079,E2 -27876.079} C_VEL
LIN {X 0,Y 140.086,Z 652.52,A -85,B 0,C 180,E1 -27879.598,E2 -27879.598} C_VEL
LIN {X 0,Y 153.075,Z 643.705,A -85,B 0,C 180,E1 -27882.304,E2 -27882.304} C_VEL
LIN {X 0,Y 165.947,Z 633.493,A -85,B 0,C 180,E1 -27884.47,E2 -27884.47} C_VEL
LIN {X 0,Y 177.615,Z 622.735,A -85,B 0,C 180,E1 -27886.155,E2 -27886.155} C_VEL
LIN {X 0,Y 188.972,Z 610.688,A -85,B 0,C 180,E1 -27887.491,E2 -27887.491} C_VEL
LIN {X 0,Y 198.989,Z 598.391,A -85,B 0,C 180,E1 -27888.549,E2 -27888.549} C_VEL
LIN {X 0,Y 209.094,Z 583.787,A -85,B 0,C 180,E1 -27889.467,E2 -27889.467} C_VEL
LIN {X 0,Y 216.692,Z 570.685,A -85,B 0,C 180,E1 -27890.117,E2 -27890.117} C_VEL
LIN {X 0,Y 224.339,Z 554.995,A -85,B 0,C 180,E1 -27890.688,E2 -27890.688} C_VEL
LIN {X 0,Y 230.198,Z 540.23,A -85,B 0,C 180,E1 -27891.098,E2 -27891.098} C_VEL
LIN {X 0,Y 235.238,Z 523.911,A -85,B 0,C 180,E1 -27891.41,E2 -27891.41} C_VEL
LIN {X 0,Y 238.816,Z 507.671,A -85,B 0,C 180,E1 -27891.69,E2 -27891.69} C_VEL
LIN {X 0,Y 240.704,Z 495.399,A -85,B 0,C 180,E1 -27891.916,E2 -27891.916} C_VEL
LIN {X 0,Y 240.64,Z 494.88,A -85,B 0,C 180,E1 -27893.292,E2 -27893.292} C_VEL
LIN {X 0,Y 240.736,Z 495.089,A -85,B 0,C 180,E1 -27895.491,E2 -27895.491} C_VEL
LIN {X 0,Y 238.106,Z 511.149,A -85,B 0,C 180,E1 -27895.763,E2 -27895.763} C_VEL
LIN {X 0,Y 234.12,Z 527.449,A -85,B 0,C 180,E1 -27896.043,E2 -27896.043} C_VEL
LIN {X 0,Y 228.997,Z 543.1,A -85,B 0,C 180,E1 -27896.531,E2 -27896.531} C_VEL
LIN {X 0,Y 222.552,Z 558.574,A -85,B 0,C 180,E1 -27897.071,E2 -27897.071} C_VEL
LIN {X 0,Y 214.503,Z 574.182,A -85,B 0,C 180,E1 -27897.847,E2 -27897.847} C_VEL
LIN {X 0,Y 205.621,Z 588.39,A -85,B 0,C 180,E1 -27898.727,E2 -27898.727} C_VEL
LIN {X 0,Y 195.854,Z 601.632,A -85,B 0,C 180,E1 -27899.799,E2 -27899.799} C_VEL
LIN {X 0,Y 184.525,Z 614.721,A -85,B 0,C 180,E1 -27901.176,E2 -27901.176} C_VEL
LIN {X 0,Y 172.406,Z 626.672,A -85,B 0,C 180,E1 -27902.886,E2 -27902.886} C_VEL
LIN {X 0,Y 160.377,Z 636.895,A -85,B 0,C 180,E1 -27904.893,E2 -27904.893} C_VEL
LIN {X 0,Y 147.092,Z 646.517,A -85,B 0,C 180,E1 -27907.51,E2 -27907.51} C_VEL
LIN {X 0,Y 135.688,Z 653.592,A -85,B 0,C 180,E1 -27910.225,E2 -27910.225} C_VEL
LIN {X 0,Y 123.116,Z 660.371,A -85,B 0,C 180,E1 -27913.965,E2 -27913.965} C_VEL
LIN {X 0,Y 111.187,Z 665.811,A -85,B 0,C 180,E1 -27918.533,E2 -27918.533} C_VEL
LIN {X 0,Y 97.925,Z 670.776,A -85,B 0,C 180,E1 -27925.509,E2 -27925.509} C_VEL
LIN {X 0,Y 90.201,Z 673.125,A -85,B 0,C 180,E1 -27931.011,E2 -27931.011} C_VEL
LIN {X 0,Y 81.768,Z 675.085,A -85,B 0,C 180,E1 -27939.325,E2 -27939.325} C_VEL
LIN {X 0,Y 75.279,Z 676.05,A -85,B 0,C 180,E1 -27949.192,E2 -27949.192} C_VEL
LIN {X 0,Y 71.082,Z 675.972,A -85,B 0,C 180,E1 -27960.372,E2 -27960.372} C_VEL
LIN {X 0,Y 69.932,Z 675.544,A -85,B 0,C 180,E1 -27966.296,E2 -27966.296} C_VEL
LIN {X 0,Y 69.047,Z 674.026,A -85,B 0,C 180,E1 -27978.253,E2 -27978.253} C_VEL
LIN {X 0,Y 70.413,Z 671.439,A -85,B 0,C 180,E1 -27989.999,E2 -27989.999} C_VEL
LIN {X 0,Y 73.146,Z 667.942,A -85,B 0,C 180,E1 -28001.078,E2 -28001.078} C_VEL
LIN {X 0,Y 77.978,Z 663.354,A -85,B 0,C 180,E1 -28011.131,E2 -28011.131} C_VEL
LIN {X 0,Y 84.575,Z 657.646,A -85,B 0,C 180,E1 -28019.906,E2 -28019.906} C_VEL
LIN {X 0,Y 92.903,Z 650.728,A -85,B 0,C 180,E1 -28027.242,E2 -28027.242} C_VEL
LIN {X 0,Y 103.605,Z 641.217,A -85,B 0,C 180,E1 -28034.051,E2 -28034.051} C_VEL
LIN {X 0,Y 114.008,Z 631.007,A -85,B 0,C 180,E1 -28039.038,E2 -28039.038} C_VEL
LIN {X 0,Y 123.671,Z 620.464,A -85,B 0,C 180,E1 -28042.711,E2 -28042.711} C_VEL
LIN {X 0,Y 133.636,Z 608.129,A -85,B 0,C 180,E1 -28045.924,E2 -28045.924} C_VEL
LIN {X 0,Y 142.45,Z 595.731,A -85,B 0,C 180,E1 -28048.326,E2 -28048.326} C_VEL
LIN {X 0,Y 150.753,Z 582.296,A -85,B 0,C 180,E1 -28050.26,E2 -28050.26} C_VEL
LIN {X 0,Y 158.334,Z 567.725,A -85,B 0,C 180,E1 -28051.908,E2 -28051.908} C_VEL
LIN {X 0,Y 164.454,Z 553.732,A -85,B 0,C 180,E1 -28053.138,E2 -28053.138} C_VEL
LIN {X 0,Y 169.955,Z 538.728,A -85,B 0,C 180,E1 -28054.08,E2 -28054.08} C_VEL
LIN {X 0,Y 174.643,Z 522.096,A -85,B 0,C 180,E1 -28054.883,E2 -28054.883} C_VEL
LIN {X 0,Y 177.988,Z 505.604,A -85,B 0,C 180,E1 -28055.409,E2 -28055.409} C_VEL
LIN {X 0,Y 181.027,Z 481.386,A -85,B 0,C 180,E1 -28055.933,E2 -28055.933} C_VEL
LIN {X 0,Y 184.58,Z 448.571,A -85,B 0,C 180,E1 -28056.677,E2 -28056.677} C_VEL
LIN {X 0,Y 182.761,Z 443.311,A -85,B 0,C 180,E1 -28059.621,E2 -28059.621} C_VEL
LIN {X 0,Y 181.142,Z 439.268,A -85,B 0,C 180,E1 -28062.802,E2 -28062.802} C_VEL
LIN {X 0,Y 180.304,Z 437.082,A -85,B 0,C 180,E1 -28064.967,E2 -28064.967} C_VEL
LIN {X 0,Y 179.537,Z 434.808,A -85,B 0,C 180,E1 -28067.787,E2 -28067.787} C_VEL
LIN {X 0,Y 178.954,Z 433.096,A -85,B 0,C 180,E1 -28073.233,E2 -28073.233} C_VEL
LIN {X 0,Y 179.281,Z 433.78,A -85,B 0,C 180,E1 -28077.309,E2 -28077.309} C_VEL
LIN {X 0,Y 179.77,Z 434.984,A -85,B 0,C 180,E1 -28079.635,E2 -28079.635} C_VEL
LIN {X 0,Y 180.907,Z 438.356,A -85,B 0,C 180,E1 -28083.183,E2 -28083.183} C_VEL
LIN {X 0,Y 182.605,Z 442.82,A -85,B 0,C 180,E1 -28086.698,E2 -28086.698} C_VEL
LIN {X 0,Y 184.582,Z 448.435,A -85,B 0,C 180,E1 -28089.918,E2 -28089.918} C_VEL
LIN {X 0,Y 184.672,Z 448.678,A -85,B 0,C 180,E1 -28090.048,E2 -28090.048} C_VEL
LIN {X 0,Y 178.14,Z 506.526,A -85,B 0,C 180,E1 -28091.322,E2 -28091.322} C_VEL
LIN {X 0,Y 174.688,Z 523.972,A -85,B 0,C 180,E1 -28091.84,E2 -28091.84} C_VEL
LIN {X 0,Y 170.079,Z 540.34,A -85,B 0,C 180,E1 -28092.519,E2 -28092.519} C_VEL
LIN {X 0,Y 164.35,Z 556.057,A -85,B 0,C 180,E1 -28093.384,E2 -28093.384} C_VEL
LIN {X 0,Y 157.94,Z 570.687,A -85,B 0,C 180,E1 -28094.574,E2 -28094.574} C_VEL
LIN {X 0,Y 150.501,Z 584.787,A -85,B 0,C 180,E1 -28095.976,E2 -28095.976} C_VEL
LIN {X 0,Y 142.114,Z 598.343,A -85,B 0,C 180,E1 -28097.83,E2 -28097.83} C_VEL
LIN {X 0,Y 132.899,Z 611.25,A -85,B 0,C 180,E1 -28100.173,E2 -28100.173} C_VEL
LIN {X 0,Y 122.507,Z 624.029,A -85,B 0,C 180,E1 -28103.381,E2 -28103.381} C_VEL
LIN {X 0,Y 112.543,Z 634.874,A -85,B 0,C 180,E1 -28107.144,E2 -28107.144} C_VEL
LIN {X 0,Y 101.86,Z 645.341,A -85,B 0,C 180,E1 -28112.306,E2 -28112.306} C_VEL
LIN {X 0,Y 92.189,Z 654.067,A -85,B 0,C 180,E1 -28118.611,E2 -28118.611} C_VEL
LIN {X 0,Y 84.76,Z 660.447,A -85,B 0,C 180,E1 -28125.188,E2 -28125.188} C_VEL
LIN {X 0,Y 77.203,Z 667.082,A -85,B 0,C 180,E1 -28135.009,E2 -28135.009} C_VEL
LIN {X 0,Y 71.954,Z 672.462,A -85,B 0,C 180,E1 -28147.003,E2 -28147.003} C_VEL
LIN {X 0,Y 69.792,Z 675.862,A -85,B 0,C 180,E1 -28158.382,E2 -28158.382} C_VEL
LIN {X 0,Y 69.73,Z 678.266,A -85,B 0,C 180,E1 -28170.001,E2 -28170.001} C_VEL
LIN {X 0,Y 69.814,Z 679.516,A -85,B 0,C 180,E1 -28181.616,E2 -28181.616} C_VEL
LIN {X 0,Y 72.047,Z 679.883,A -85,B 0,C 180,E1 -28192.967,E2 -28192.967} C_VEL
LIN {X 0,Y 78.833,Z 678.862,A -85,B 0,C 180,E1 -28206.649,E2 -28206.649} C_VEL
LIN {X 0,Y 87.526,Z 676.616,A -85,B 0,C 180,E1 -28216.276,E2 -28216.276} C_VEL
LIN {X 0,Y 91.28,Z 675.444,A -85,B 0,C 180,E1 -28219.397,E2 -28219.397} C_VEL
LIN {X 0,Y 94.541,Z 674.295,A -85,B 0,C 180,E1 -28222.354,E2 -28222.354} C_VEL
LIN {X 0,Y 99.065,Z 672.173,A -85,B 0,C 180,E1 -28227.429,E2 -28227.429} C_VEL
LIN {X 0,Y 103.047,Z 670.173,A -85,B 0,C 180,E1 -28231.157,E2 -28231.157} C_VEL
LIN {X 0,Y 106.816,Z 668.432,A -85,B 0,C 180,E1 -28233.453,E2 -28233.453} C_VEL
LIN {X 0,Y 108.271,Z 667.788,A -85,B 0,C 180,E1 -28234.075,E2 -28234.075} C_VEL
LIN {X 0,Y 121.051,Z 662,A -85,B 0,C 180,E1 -28238.27,E2 -28238.27} C_VEL
LIN {X 0,Y 136.357,Z 653.635,A -85,B 0,C 180,E1 -28242.084,E2 -28242.084} C_VEL
LIN {X 0,Y 151.061,Z 644.016,A -85,B 0,C 180,E1 -28244.88,E2 -28244.88} C_VEL
LIN {X 0,Y 164.189,Z 633.886,A -85,B 0,C 180,E1 -28246.857,E2 -28246.857} C_VEL
LIN {X 0,Y 175.765,Z 623.529,A -85,B 0,C 180,E1 -28248.356,E2 -28248.356} C_VEL
LIN {X 0,Y 185.886,Z 613.252,A -85,B 0,C 180,E1 -28249.426,E2 -28249.426} C_VEL
LIN {X 0,Y 195.187,Z 602.335,A -85,B 0,C 180,E1 -28250.294,E2 -28250.294} C_VEL
LIN {X 0,Y 203.668,Z 591.087,A -85,B 0,C 180,E1 -28251.03,E2 -28251.03} C_VEL
LIN {X 0,Y 213.033,Z 576.43,A -85,B 0,C 180,E1 -28251.774,E2 -28251.774} C_VEL
LIN {X 0,Y 220.735,Z 561.987,A -85,B 0,C 180,E1 -28252.306,E2 -28252.306} C_VEL
LIN {X 0,Y 227.604,Z 546.324,A -85,B 0,C 180,E1 -28252.731,E2 -28252.731} C_VEL
LIN {X 0,Y 233.053,Z 530.686,A -85,B 0,C 180,E1 -28253.052,E2 -28253.052} C_VEL
LIN {X 0,Y 237.363,Z 514.204,A -85,B 0,C 180,E1 -28253.292,E2 -28253.292} C_VEL
LIN {X 0,Y 239.613,Z 501.924,A -85,B 0,C 180,E1 -28253.513,E2 -28253.513} C_VEL
LIN {X 0,Y 239.592,Z 502.048,A -85,B 0,C 180,E1 -28253.928,E2 -28253.928} C_VEL
LIN {X 0,Y 236.257,Z 518.751,A -85,B 0,C 180,E1 -28254.167,E2 -28254.167} C_VEL
LIN {X 0,Y 232.24,Z 533.208,A -85,B 0,C 180,E1 -28254.441,E2 -28254.441} C_VEL
LIN {X 0,Y 226.473,Z 549.087,A -85,B 0,C 180,E1 -28254.927,E2 -28254.927} C_VEL
LIN {X 0,Y 220.335,Z 562.573,A -85,B 0,C 180,E1 -28255.402,E2 -28255.402} C_VEL
LIN {X 0,Y 212.212,Z 577.474,A -85,B 0,C 180,E1 -28256.096,E2 -28256.096} C_VEL
LIN {X 0,Y 203.232,Z 591.277,A -85,B 0,C 180,E1 -28256.899,E2 -28256.899} C_VEL
LIN {X 0,Y 193.305,Z 604.177,A -85,B 0,C 180,E1 -28257.918,E2 -28257.918} C_VEL
LIN {X 0,Y 182.753,Z 615.907,A -85,B 0,C 180,E1 -28259.063,E2 -28259.063} C_VEL
LIN {X 0,Y 170.347,Z 627.776,A -85,B 0,C 180,E1 -28260.644,E2 -28260.644} C_VEL
LIN {X 0,Y 157.769,Z 638.083,A -85,B 0,C 180,E1 -28262.555,E2 -28262.555} C_VEL
LIN {X 0,Y 144.607,Z 647.319,A -85,B 0,C 180,E1 -28264.914,E2 -28264.914} C_VEL
LIN {X 0,Y 131.249,Z 655.222,A -85,B 0,C 180,E1 -28267.85,E2 -28267.85} C_VEL
LIN {X 0,Y 118.326,Z 661.695,A -85,B 0,C 180,E1 -28271.47,E2 -28271.47} C_VEL
LIN {X 0,Y 108.319,Z 666.015,A -85,B 0,C 180,E1 -28275.044,E2 -28275.044} C_VEL
LIN {X 0,Y 97.263,Z 669.998,A -85,B 0,C 180,E1 -28280.056,E2 -28280.056} C_VEL
LIN {X 0,Y 86.545,Z 673.186,A -85,B 0,C 180,E1 -28286.712,E2 -28286.712} C_VEL
LIN {X 0,Y 77.194,Z 675.202,A -85,B 0,C 180,E1 -28294.975,E2 -28294.975} C_VEL
LIN {X 0,Y 69.759,Z 676.249,A -85,B 0,C 180,E1 -28305.151,E2 -28305.151} C_VEL
LIN {X 0,Y 64.674,Z 676.211,A -85,B 0,C 180,E1 -28317.088,E2 -28317.088} C_VEL
LIN {X 0,Y 63.205,Z 675.822,A -85,B 0,C 180,E1 -28323.59,E2 -28323.59} C_VEL
LIN {X 0,Y 61.944,Z 674.364,A -85,B 0,C 180,E1 -28336.884,E2 -28336.884} C_VEL
LIN {X 0,Y 63.256,Z 671.826,A -85,B 0,C 180,E1 -28349.999,E2 -28349.999} C_VEL
LIN {X 0,Y 66.18,Z 668.41,A -85,B 0,C 180,E1 -28362.262,E2 -28362.262} C_VEL
LIN {X 0,Y 71.408,Z 663.863,A -85,B 0,C 180,E1 -28373.183,E2 -28373.183} C_VEL
LIN {X 0,Y 78.51,Z 658.245,A -85,B 0,C 180,E1 -28382.486,E2 -28382.486} C_VEL
LIN {X 0,Y 87.366,Z 651.389,A -85,B 0,C 180,E1 -28390.056,E2 -28390.056} C_VEL
LIN {X 0,Y 97.328,Z 643.082,A -85,B 0,C 180,E1 -28396.227,E2 -28396.227} C_VEL
LIN {X 0,Y 108.116,Z 633.215,A -85,B 0,C 180,E1 -28401.264,E2 -28401.264} C_VEL
LIN {X 0,Y 118.086,Z 623.072,A -85,B 0,C 180,E1 -28404.919,E2 -28404.919} C_VEL
LIN {X 0,Y 128.336,Z 611.199,A -85,B 0,C 180,E1 -28408.083,E2 -28408.083} C_VEL
LIN {X 0,Y 138.866,Z 597.06,A -85,B 0,C 180,E1 -28410.811,E2 -28410.811} C_VEL
LIN {X 0,Y 148.171,Z 582.469,A -85,B 0,C 180,E1 -28412.79,E2 -28412.79} C_VEL
LIN {X 0,Y 155.931,Z 567.896,A -85,B 0,C 180,E1 -28414.346,E2 -28414.346} C_VEL
LIN {X 0,Y 162.199,Z 553.888,A -85,B 0,C 180,E1 -28415.494,E2 -28415.494} C_VEL
LIN {X 0,Y 167.805,Z 538.872,A -85,B 0,C 180,E1 -28416.371,E2 -28416.371} C_VEL
LIN {X 0,Y 172.583,Z 522.233,A -85,B 0,C 180,E1 -28417.123,E2 -28417.123} C_VEL
LIN {X 0,Y 175.912,Z 506.164,A -85,B 0,C 180,E1 -28417.594,E2 -28417.594} C_VEL
LIN {X 0,Y 178.835,Z 483.666,A -85,B 0,C 180,E1 -28418.06,E2 -28418.06} C_VEL
LIN {X 0,Y 182.266,Z 452.626,A -85,B 0,C 180,E1 -28418.736,E2 -28418.736} C_VEL
LIN {X 0,Y 180.843,Z 448.421,A -85,B 0,C 180,E1 -28421.404,E2 -28421.404} C_VEL
LIN {X 0,Y 179.283,Z 444.082,A -85,B 0,C 180,E1 -28425.287,E2 -28425.287} C_VEL
LIN {X 0,Y 178.536,Z 441.73,A -85,B 0,C 180,E1 -28428.277,E2 -28428.277} C_VEL
LIN {X 0,Y 178.076,Z 440.166,A -85,B 0,C 180,E1 -28433.199,E2 -28433.199} C_VEL
LIN {X 0,Y 178.328,Z 440.691,A -85,B 0,C 180,E1 -28436.848,E2 -28436.848} C_VEL
LIN {X 0,Y 178.772,Z 441.997,A -85,B 0,C 180,E1 -28439.266,E2 -28439.266} C_VEL
LIN {X 0,Y 179.741,Z 445.143,A -85,B 0,C 180,E1 -28442.59,E2 -28442.59} C_VEL
LIN {X 0,Y 181.154,Z 449.203,A -85,B 0,C 180,E1 -28445.813,E2 -28445.813} C_VEL
LIN {X 0,Y 182.34,Z 452.735,A -85,B 0,C 180,E1 -28447.987,E2 -28447.987} C_VEL
LIN {X 0,Y 176.246,Z 505.724,A -85,B 0,C 180,E1 -28449.103,E2 -28449.103} C_VEL
LIN {X 0,Y 172.848,Z 522.874,A -85,B 0,C 180,E1 -28449.576,E2 -28449.576} C_VEL
LIN {X 0,Y 168.255,Z 539.233,A -85,B 0,C 180,E1 -28450.198,E2 -28450.198} C_VEL
LIN {X 0,Y 162.427,Z 555.163,A -85,B 0,C 180,E1 -28450.991,E2 -28450.991} C_VEL
LIN {X 0,Y 156.273,Z 569.108,A -85,B 0,C 180,E1 -28452,E2 -28452} C_VEL
LIN {X 0,Y 148.109,Z 584.378,A -85,B 0,C 180,E1 -28453.405,E2 -28453.405} C_VEL
LIN {X 0,Y 139.89,Z 597.38,A -85,B 0,C 180,E1 -28455.042,E2 -28455.042} C_VEL
LIN {X 0,Y 130.573,Z 610.195,A -85,B 0,C 180,E1 -28457.181,E2 -28457.181} C_VEL
LIN {X 0,Y 121.339,Z 621.45,A -85,B 0,C 180,E1 -28459.746,E2 -28459.746} C_VEL
LIN {X 0,Y 110.884,Z 632.617,A -85,B 0,C 180,E1 -28463.216,E2 -28463.216} C_VEL
LIN {X 0,Y 99.544,Z 643.385,A -85,B 0,C 180,E1 -28468.053,E2 -28468.053} C_VEL
LIN {X 0,Y 88.865,Z 652.557,A -85,B 0,C 180,E1 -28474.197,E2 -28474.197} C_VEL
LIN {X 0,Y 79.784,Z 659.889,A -85,B 0,C 180,E1 -28481.519,E2 -28481.519} C_VEL
LIN {X 0,Y 71.903,Z 666.207,A -85,B 0,C 180,E1 -28490.918,E2 -28490.918} C_VEL
LIN {X 0,Y 65.411,Z 672.037,A -85,B 0,C 180,E1 -28504.547,E2 -28504.547} C_VEL
LIN {X 0,Y 62.805,Z 675.499,A -85,B 0,C 180,E1 -28517.068,E2 -28517.068} C_VEL
LIN {X 0,Y 62.623,Z 677.972,A -85,B 0,C 180,E1 -28530.001,E2 -28530.001} C_VEL
LIN {X 0,Y 62.83,Z 679.256,A -85,B 0,C 180,E1 -28542.928,E2 -28542.928} C_VEL
LIN {X 0,Y 65.509,Z 679.677,A -85,B 0,C 180,E1 -28555.413,E2 -28555.413} C_VEL
LIN {X 0,Y 72.754,Z 678.782,A -85,B 0,C 180,E1 -28569.399,E2 -28569.399} C_VEL
LIN {X 0,Y 82.722,Z 676.526,A -85,B 0,C 180,E1 -28579.875,E2 -28579.875} C_VEL
LIN {X 0,Y 92.502,Z 673.659,A -85,B 0,C 180,E1 -28586.695,E2 -28586.695} C_VEL
LIN {X 0,Y 106.229,Z 668.67,A -85,B 0,C 180,E1 -28593.272,E2 -28593.272} C_VEL
LIN {X 0,Y 108.271,Z 667.788,A -85,B 0,C 180,E1 -28594.075,E2 -28594.075} C_VEL
LIN {X 0,Y 112.458,Z 665.896,A -85,B 0,C 180,E1 -28596.004,E2 -28596.004} C_VEL
LIN {X 0,Y 118.567,Z 662.655,A -85,B 0,C 180,E1 -28599.549,E2 -28599.549} C_VEL
LIN {X 0,Y 124.958,Z 659.072,A -85,B 0,C 180,E1 -28602.69,E2 -28602.69} C_VEL
LIN {X 0,Y 129.431,Z 656.561,A -85,B 0,C 180,E1 -28604.007,E2 -28604.007} C_VEL
LIN {X 0,Y 142.76,Z 648.722,A -85,B 0,C 180,E1 -28606.481,E2 -28606.481} C_VEL
LIN {X 0,Y 156.022,Z 639.502,A -85,B 0,C 180,E1 -28608.445,E2 -28608.445} C_VEL
LIN {X 0,Y 167.778,Z 630.062,A -85,B 0,C 180,E1 -28609.863,E2 -28609.863} C_VEL
LIN {X 0,Y 179.601,Z 619.131,A -85,B 0,C 180,E1 -28611.139,E2 -28611.139} C_VEL
LIN {X 0,Y 191.541,Z 606.217,A -85,B 0,C 180,E1 -28612.175,E2 -28612.175} C_VEL
LIN {X 0,Y 201.827,Z 593.092,A -85,B 0,C 180,E1 -28612.944,E2 -28612.944} C_VEL
LIN {X 0,Y 211.289,Z 578.873,A -85,B 0,C 180,E1 -28613.592,E2 -28613.592} C_VEL
LIN {X 0,Y 214.151,Z 574.1,A -85,B 0,C 180,E1 -28613.781,E2 -28613.781} C_VEL
LIN {X 0,Y 214.588,Z 573.298,A -85,B 0,C 180,E1 -28613.983,E2 -28613.983} C_VEL
LIN {X 0,Y 206.152,Z 586.792,A -85,B 0,C 180,E1 -28614.638,E2 -28614.638} C_VEL
LIN {X 0,Y 197.431,Z 598.8,A -85,B 0,C 180,E1 -28615.364,E2 -28615.364} C_VEL
LIN {X 0,Y 186.615,Z 611.492,A -85,B 0,C 180,E1 -28616.382,E2 -28616.382} C_VEL
LIN {X 0,Y 175.869,Z 622.309,A -85,B 0,C 180,E1 -28617.498,E2 -28617.498} C_VEL
LIN {X 0,Y 163.426,Z 633.149,A -85,B 0,C 180,E1 -28619.02,E2 -28619.02} C_VEL
LIN {X 0,Y 151.117,Z 642.391,A -85,B 0,C 180,E1 -28620.79,E2 -28620.79} C_VEL
LIN {X 0,Y 136.331,Z 651.752,A -85,B 0,C 180,E1 -28623.381,E2 -28623.381} C_VEL
LIN {X 0,Y 121.526,Z 659.516,A -85,B 0,C 180,E1 -28626.644,E2 -28626.644} C_VEL
LIN {X 0,Y 107.337,Z 665.633,A -85,B 0,C 180,E1 -28630.841,E2 -28630.841} C_VEL
LIN {X 0,Y 94.931,Z 669.997,A -85,B 0,C 180,E1 -28635.755,E2 -28635.755} C_VEL
LIN {X 0,Y 83.406,Z 673.227,A -85,B 0,C 180,E1 -28642.044,E2 -28642.044} C_VEL
LIN {X 0,Y 73.124,Z 675.32,A -85,B 0,C 180,E1 -28650.116,E2 -28650.116} C_VEL
LIN {X 0,Y 64.259,Z 676.46,A -85,B 0,C 180,E1 -28661.017,E2 -28661.017} C_VEL
LIN {X 0,Y 58.536,Z 676.449,A -85,B 0,C 180,E1 -28673.107,E2 -28673.107} C_VEL
LIN {X 0,Y 55.403,Z 675.527,A -85,B 0,C 180,E1 -28687.631,E2 -28687.631} C_VEL
LIN {X 0,Y 55.055,Z 673.563,A -85,B 0,C 180,E1 -28702.665,E2 -28702.665} C_VEL
LIN {X 0,Y 56.237,Z 672.002,A -85,B 0,C 180,E1 -28711.026,E2 -28711.026} C_VEL
LIN {X 0,Y 59.251,Z 668.863,A -85,B 0,C 180,E1 -28723.722,E2 -28723.722} C_VEL
LIN {X 0,Y 64.951,Z 664.372,A -85,B 0,C 180,E1 -28735.646,E2 -28735.646} C_VEL
LIN {X 0,Y 72.634,Z 658.844,A -85,B 0,C 180,E1 -28745.489,E2 -28745.489} C_VEL
LIN {X 0,Y 82.065,Z 652.036,A -85,B 0,C 180,E1 -28753.244,E2 -28753.244} C_VEL
LIN {X 0,Y 92.581,Z 643.83,A -85,B 0,C 180,E1 -28759.386,E2 -28759.386} C_VEL
LIN {X 0,Y 103.843,Z 634.079,A -85,B 0,C 180,E1 -28764.306,E2 -28764.306} C_VEL
LIN {X 0,Y 114.171,Z 624.069,A -85,B 0,C 180,E1 -28767.822,E2 -28767.822} C_VEL
LIN {X 0,Y 124.744,Z 612.277,A -85,B 0,C 180,E1 -28770.839,E2 -28770.839} C_VEL
LIN {X 0,Y 134.025,Z 600.412,A -85,B 0,C 180,E1 -28773.055,E2 -28773.055} C_VEL
LIN {X 0,Y 143.475,Z 586.481,A -85,B 0,C 180,E1 -28774.986,E2 -28774.986} C_VEL
LIN {X 0,Y 151.453,Z 572.71,A -85,B 0,C 180,E1 -28776.415,E2 -28776.415} C_VEL
LIN {X 0,Y 158.616,Z 557.839,A -85,B 0,C 180,E1 -28777.658,E2 -28777.658} C_VEL
LIN {X 0,Y 164.702,Z 542.413,A -85,B 0,C 180,E1 -28778.553,E2 -28778.553} C_VEL
LIN {X 0,Y 169.776,Z 526.014,A -85,B 0,C 180,E1 -28779.274,E2 -28779.274} C_VEL
LIN {X 0,Y 173.647,Z 508.999,A -85,B 0,C 180,E1 -28779.773,E2 -28779.773} C_VEL
LIN {X 0,Y 176.358,Z 490.343,A -85,B 0,C 180,E1 -28780.154,E2 -28780.154} C_VEL
LIN {X 0,Y 180.149,Z 456.856,A -85,B 0,C 180,E1 -28780.84,E2 -28780.84} C_VEL
LIN {X 0,Y 178.721,Z 452.552,A -85,B 0,C 180,E1 -28784.195,E2 -28784.195} C_VEL
LIN {X 0,Y 177.983,Z 450.252,A -85,B 0,C 180,E1 -28786.623,E2 -28786.623} C_VEL
LIN {X 0,Y 177.585,Z 448.71,A -85,B 0,C 180,E1 -28788.586,E2 -28788.586} C_VEL
LIN {X 0,Y 177.197,Z 447.241,A -85,B 0,C 180,E1 -28793.165,E2 -28793.165} C_VEL
LIN {X 0,Y 177.399,Z 447.649,A -85,B 0,C 180,E1 -28796.488,E2 -28796.488} C_VEL
LIN {X 0,Y 177.801,Z 449.022,A -85,B 0,C 180,E1 -28798.964,E2 -28798.964} C_VEL
LIN {X 0,Y 178.652,Z 452.056,A -85,B 0,C 180,E1 -28802.144,E2 -28802.144} C_VEL
LIN {X 0,Y 179.817,Z 455.8,A -85,B 0,C 180,E1 -28805.069,E2 -28805.069} C_VEL
LIN {X 0,Y 180.207,Z 457.1,A -85,B 0,C 180,E1 -28805.898,E2 -28805.898} C_VEL
LIN {X 0,Y 174.346,Z 506.458,A -85,B 0,C 180,E1 -28806.873,E2 -28806.873} C_VEL
LIN {X 0,Y 170.852,Z 523.545,A -85,B 0,C 180,E1 -28807.31,E2 -28807.31} C_VEL
LIN {X 0,Y 165.851,Z 540.668,A -85,B 0,C 180,E1 -28807.895,E2 -28807.895} C_VEL
LIN {X 0,Y 160.366,Z 555.228,A -85,B 0,C 180,E1 -28808.585,E2 -28808.585} C_VEL
LIN {X 0,Y 153.268,Z 570.748,A -85,B 0,C 180,E1 -28809.644,E2 -28809.644} C_VEL
LIN {X 0,Y 145.775,Z 584.376,A -85,B 0,C 180,E1 -28810.796,E2 -28810.796} C_VEL
LIN {X 0,Y 137.952,Z 596.479,A -85,B 0,C 180,E1 -28812.168,E2 -28812.168} C_VEL
LIN {X 0,Y 128.621,Z 609.143,A -85,B 0,C 180,E1 -28814.099,E2 -28814.099} C_VEL
LIN {X 0,Y 119.077,Z 620.512,A -85,B 0,C 180,E1 -28816.447,E2 -28816.447} C_VEL
LIN {X 0,Y 108.234,Z 631.765,A -85,B 0,C 180,E1 -28819.69,E2 -28819.69} C_VEL
LIN {X 0,Y 97.797,Z 641.379,A -85,B 0,C 180,E1 -28823.616,E2 -28823.616} C_VEL
LIN {X 0,Y 86.609,Z 650.638,A -85,B 0,C 180,E1 -28829.133,E2 -28829.133} C_VEL
LIN {X 0,Y 77.571,Z 657.566,A -85,B 0,C 180,E1 -28835.373,E2 -28835.373} C_VEL
LIN {X 0,Y 68.609,Z 664.088,A -85,B 0,C 180,E1 -28844.189,E2 -28844.189} C_VEL
LIN {X 0,Y 61.594,Z 669.413,A -85,B 0,C 180,E1 -28855.215,E2 -28855.215} C_VEL
LIN {X 0,Y 57.037,Z 673.492,A -85,B 0,C 180,E1 -28868.307,E2 -28868.307} C_VEL
LIN {X 0,Y 55.361,Z 676.53,A -85,B 0,C 180,E1 -28882.707,E2 -28882.707} C_VEL
LIN {X 0,Y 55.51,Z 677.657,A -85,B 0,C 180,E1 -28890.001,E2 -28890.001} C_VEL
LIN {X 0,Y 55.898,Z 678.996,A -85,B 0,C 180,E1 -28904.565,E2 -28904.565} C_VEL
LIN {X 0,Y 59.119,Z 679.452,A -85,B 0,C 180,E1 -28918.394,E2 -28918.394} C_VEL
LIN {X 0,Y 66.876,Z 678.688,A -85,B 0,C 180,E1 -28932.644,E2 -28932.644} C_VEL
LIN {X 0,Y 78.279,Z 676.439,A -85,B 0,C 180,E1 -28943.905,E2 -28943.905} C_VEL
LIN {X 0,Y 88.753,Z 673.65,A -85,B 0,C 180,E1 -28950.581,E2 -28950.581} C_VEL
LIN {X 0,Y 103.197,Z 668.716,A -85,B 0,C 180,E1 -28956.838,E2 -28956.838} C_VEL
LIN {X 0,Y 118.594,Z 662.113,A -85,B 0,C 180,E1 -28961.475,E2 -28961.475} C_VEL
LIN {X 0,Y 129.431,Z 656.561,A -85,B 0,C 180,E1 -28964.007,E2 -28964.007} C_VEL
LIN {X 0,Y 133.937,Z 653.976,A -85,B 0,C 180,E1 -28965.231,E2 -28965.231} C_VEL
LIN {X 0,Y 147.481,Z 645.035,A -85,B 0,C 180,E1 -28969.89,E2 -28969.89} C_VEL
LIN {X 0,Y 151.965,Z 641.853,A -85,B 0,C 180,E1 -28970.698,E2 -28970.698} C_VEL
LIN {X 0,Y 164.97,Z 631.977,A -85,B 0,C 180,E1 -28972.095,E2 -28972.095} C_VEL
LIN {X 0,Y 176.931,Z 621.299,A -85,B 0,C 180,E1 -28973.239,E2 -28973.239} C_VEL
LIN {X 0,Y 185.532,Z 612.655,A -85,B 0,C 180,E1 -28973.878,E2 -28973.878} C_VEL
LIN {X 0,Y 186.502,Z 611.565,A -85,B 0,C 180,E1 -28974.168,E2 -28974.168} C_VEL
LIN {X 0,Y 174.411,Z 623.532,A -85,B 0,C 180,E1 -28975.262,E2 -28975.262} C_VEL
LIN {X 0,Y 161.929,Z 634.098,A -85,B 0,C 180,E1 -28976.603,E2 -28976.603} C_VEL
LIN {X 0,Y 149.421,Z 643.22,A -85,B 0,C 180,E1 -28978.183,E2 -28978.183} C_VEL
LIN {X 0,Y 135.443,Z 651.859,A -85,B 0,C 180,E1 -28980.332,E2 -28980.332} C_VEL
LIN {X 0,Y 123.119,Z 658.265,A -85,B 0,C 180,E1 -28982.611,E2 -28982.611} C_VEL
LIN {X 0,Y 109.509,Z 664.278,A -85,B 0,C 180,E1 -28985.868,E2 -28985.868} C_VEL
LIN {X 0,Y 96.354,Z 668.994,A -85,B 0,C 180,E1 -28990.037,E2 -28990.037} C_VEL
LIN {X 0,Y 86.672,Z 671.862,A -85,B 0,C 180,E1 -28994.082,E2 -28994.082} C_VEL
LIN {X 0,Y 71.663,Z 675.146,A -85,B 0,C 180,E1 -29003.1,E2 -29003.1} C_VEL
LIN {X 0,Y 60.006,Z 676.611,A -85,B 0,C 180,E1 -29014.928,E2 -29014.928} C_VEL
LIN {X 0,Y 52.736,Z 676.688,A -85,B 0,C 180,E1 -29028.214,E2 -29028.214} C_VEL
LIN {X 0,Y 48.643,Z 675.839,A -85,B 0,C 180,E1 -29044.313,E2 -29044.313} C_VEL
LIN {X 0,Y 47.846,Z 673.915,A -85,B 0,C 180,E1 -29061.552,E2 -29061.552} C_VEL
LIN {X 0,Y 49.243,Z 672.172,A -85,B 0,C 180,E1 -29072.385,E2 -29072.385} C_VEL
LIN {X 0,Y 53.702,Z 668.277,A -85,B 0,C 180,E1 -29089.097,E2 -29089.097} C_VEL
LIN {X 0,Y 60.58,Z 663.642,A -85,B 0,C 180,E1 -29101.469,E2 -29101.469} C_VEL
LIN {X 0,Y 69.422,Z 657.831,A -85,B 0,C 180,E1 -29111.149,E2 -29111.149} C_VEL
LIN {X 0,Y 81.138,Z 649.804,A -85,B 0,C 180,E1 -29119.279,E2 -29119.279} C_VEL
LIN {X 0,Y 92.492,Z 641.181,A -85,B 0,C 180,E1 -29124.768,E2 -29124.768} C_VEL
LIN {X 0,Y 104.412,Z 630.889,A -85,B 0,C 180,E1 -29129.115,E2 -29129.115} C_VEL
LIN {X 0,Y 115.202,Z 620.197,A -85,B 0,C 180,E1 -29132.2,E2 -29132.2} C_VEL
LIN {X 0,Y 126.212,Z 607.67,A -85,B 0,C 180,E1 -29134.805,E2 -29134.805} C_VEL
LIN {X 0,Y 136.578,Z 593.889,A -85,B 0,C 180,E1 -29136.897,E2 -29136.897} C_VEL
LIN {X 0,Y 145.525,Z 579.998,A -85,B 0,C 180,E1 -29138.382,E2 -29138.382} C_VEL
LIN {X 0,Y 152.825,Z 566.566,A -85,B 0,C 180,E1 -29139.551,E2 -29139.551} C_VEL
LIN {X 0,Y 159.375,Z 552.084,A -85,B 0,C 180,E1 -29140.489,E2 -29140.489} C_VEL
LIN {X 0,Y 165.173,Z 536.381,A -85,B 0,C 180,E1 -29141.212,E2 -29141.212} C_VEL
LIN {X 0,Y 169.699,Z 520.466,A -85,B 0,C 180,E1 -29141.794,E2 -29141.794} C_VEL
LIN {X 0,Y 173.006,Z 504.404,A -85,B 0,C 180,E1 -29142.173,E2 -29142.173} C_VEL
LIN {X 0,Y 178.166,Z 462.275,A -85,B 0,C 180,E1 -29142.92,E2 -29142.92} C_VEL
LIN {X 0,Y 178.212,Z 461.412,A -85,B 0,C 180,E1 -29143.033,E2 -29143.033} C_VEL
LIN {X 0,Y 177.085,Z 457.534,A -85,B 0,C 180,E1 -29146.585,E2 -29146.585} C_VEL
LIN {X 0,Y 176.58,Z 455.577,A -85,B 0,C 180,E1 -29149.233,E2 -29149.233} C_VEL
LIN {X 0,Y 176.319,Z 454.307,A -85,B 0,C 180,E1 -29153.131,E2 -29153.131} C_VEL
LIN {X 0,Y 176.513,Z 454.742,A -85,B 0,C 180,E1 -29156.47,E2 -29156.47} C_VEL
LIN {X 0,Y 176.793,Z 455.87,A -85,B 0,C 180,E1 -29158.428,E2 -29158.428} C_VEL
LIN {X 0,Y 177.512,Z 458.791,A -85,B 0,C 180,E1 -29161.501,E2 -29161.501} C_VEL
LIN {X 0,Y 178.273,Z 461.583,A -85,B 0,C 180,E1 -29163.725,E2 -29163.725} C_VEL
LIN {X 0,Y 172.851,Z 506.334,A -85,B 0,C 180,E1 -29164.59,E2 -29164.59} C_VEL
LIN {X 0,Y 169.309,Z 523.377,A -85,B 0,C 180,E1 -29164.975,E2 -29164.975} C_VEL
LIN {X 0,Y 164.592,Z 539.453,A -85,B 0,C 180,E1 -29165.482,E2 -29165.482} C_VEL
LIN {X 0,Y 158.595,Z 555.247,A -85,B 0,C 180,E1 -29166.122,E2 -29166.122} C_VEL
LIN {X 0,Y 151.374,Z 570.718,A -85,B 0,C 180,E1 -29167.07,E2 -29167.07} C_VEL
LIN {X 0,Y 143.754,Z 584.322,A -85,B 0,C 180,E1 -29168.109,E2 -29168.109} C_VEL
LIN {X 0,Y 135.352,Z 597.008,A -85,B 0,C 180,E1 -29169.407,E2 -29169.407} C_VEL
LIN {X 0,Y 127.06,Z 608.059,A -85,B 0,C 180,E1 -29170.952,E2 -29170.952} C_VEL
LIN {X 0,Y 117.227,Z 619.503,A -85,B 0,C 180,E1 -29173.039,E2 -29173.039} C_VEL
LIN {X 0,Y 106.019,Z 630.9,A -85,B 0,C 180,E1 -29176.014,E2 -29176.014} C_VEL
LIN {X 0,Y 95.125,Z 640.628,A -85,B 0,C 180,E1 -29179.613,E2 -29179.613} C_VEL
LIN {X 0,Y 84.686,Z 648.984,A -85,B 0,C 180,E1 -29184.096,E2 -29184.096} C_VEL
LIN {X 0,Y 73.611,Z 656.964,A -85,B 0,C 180,E1 -29190.766,E2 -29190.766} C_VEL
LIN {X 0,Y 63.784,Z 663.571,A -85,B 0,C 180,E1 -29199.531,E2 -29199.531} C_VEL
LIN {X 0,Y 55.824,Z 668.961,A -85,B 0,C 180,E1 -29210.989,E2 -29210.989} C_VEL
LIN {X 0,Y 50.43,Z 673.091,A -85,B 0,C 180,E1 -29225.287,E2 -29225.287} C_VEL
LIN {X 0,Y 48.299,Z 676.203,A -85,B 0,C 180,E1 -29241.634,E2 -29241.634} C_VEL
LIN {X 0,Y 48.416,Z 677.332,A -85,B 0,C 180,E1 -29250.001,E2 -29250.001} C_VEL
LIN {X 0,Y 49.002,Z 678.736,A -85,B 0,C 180,E1 -29266.67,E2 -29266.67} C_VEL
LIN {X 0,Y 52.93,Z 679.225,A -85,B 0,C 180,E1 -29282.082,E2 -29282.082} C_VEL
LIN {X 0,Y 61.169,Z 678.606,A -85,B 0,C 180,E1 -29296.425,E2 -29296.425} C_VEL
LIN {X 0,Y 69.083,Z 677.399,A -85,B 0,C 180,E1 -29304.476,E2 -29304.476} C_VEL
LIN {X 0,Y 79.731,Z 675.103,A -85,B 0,C 180,E1 -29311.82,E2 -29311.82} C_VEL
LIN {X 0,Y 91.691,Z 671.743,A -85,B 0,C 180,E1 -29317.468,E2 -29317.468} C_VEL
LIN {X 0,Y 103.721,Z 667.566,A -85,B 0,C 180,E1 -29321.555,E2 -29321.555} C_VEL
LIN {X 0,Y 116.523,Z 662.222,A -85,B 0,C 180,E1 -29324.805,E2 -29324.805} C_VEL
LIN {X 0,Y 129.937,Z 655.508,A -85,B 0,C 180,E1 -29327.507,E2 -29327.507} C_VEL
LIN {X 0,Y 144.624,Z 646.809,A -85,B 0,C 180,E1 -29329.755,E2 -29329.755} C_VEL
LIN {X 0,Y 151.965,Z 641.853,A -85,B 0,C 180,E1 -29330.698,E2 -29330.698} C_VEL
LIN {X 0,Y 152.418,Z 641.464,A -85,B 0,C 180,E1 -29331.142,E2 -29331.142} C_VEL
LIN {X 0,Y 151.635,Z 641.875,A -85,B 0,C 180,E1 -29332.078,E2 -29332.078} C_VEL
LIN {X 0,Y 148.415,Z 643.894,A -85,B 0,C 180,E1 -29333.593,E2 -29333.593} C_VEL
LIN {X 0,Y 143.179,Z 647.15,A -85,B 0,C 180,E1 -29335.091,E2 -29335.091} C_VEL
LIN {X 0,Y 139.026,Z 649.604,A -85,B 0,C 180,E1 -29336.162,E2 -29336.162} C_VEL
LIN {X 0,Y 132.469,Z 653.307,A -85,B 0,C 180,E1 -29337.563,E2 -29337.563} C_VEL
LIN {X 0,Y 130.172,Z 654.504,A -85,B 0,C 180,E1 -29337.944,E2 -29337.944} C_VEL
LIN {X 0,Y 115.246,Z 661.596,A -85,B 0,C 180,E1 -29340.558,E2 -29340.558} C_VEL
LIN {X 0,Y 100.603,Z 667.262,A -85,B 0,C 180,E1 -29344.008,E2 -29344.008} C_VEL
LIN {X 0,Y 85.395,Z 671.802,A -85,B 0,C 180,E1 -29349.03,E2 -29349.03} C_VEL
LIN {X 0,Y 72.764,Z 674.56,A -85,B 0,C 180,E1 -29355.011,E2 -29355.011} C_VEL
LIN {X 0,Y 61.207,Z 676.325,A -85,B 0,C 180,E1 -29363.277,E2 -29363.277} C_VEL
LIN {X 0,Y 51.379,Z 676.966,A -85,B 0,C 180,E1 -29374.842,E2 -29374.842} C_VEL
LIN {X 0,Y 43.336,Z 676.444,A -85,B 0,C 180,E1 -29394.19,E2 -29394.19} C_VEL
LIN {X 0,Y 40.844,Z 675.304,A -85,B 0,C 180,E1 -29409.87,E2 -29409.87} C_VEL
LIN {X 0,Y 41.553,Z 672.995,A -85,B 0,C 180,E1 -29429.999,E2 -29429.999} C_VEL
LIN {X 0,Y 43.238,Z 671.503,A -85,B 0,C 180,E1 -29439.353,E2 -29439.353} C_VEL
LIN {X 0,Y 50.577,Z 666.598,A -85,B 0,C 180,E1 -29459.1,E2 -29459.1} C_VEL
LIN {X 0,Y 61.654,Z 660.003,A -85,B 0,C 180,E1 -29473.152,E2 -29473.152} C_VEL
LIN {X 0,Y 75.264,Z 651.482,A -85,B 0,C 180,E1 -29482.533,E2 -29482.533} C_VEL
LIN {X 0,Y 88.592,Z 641.953,A -85,B 0,C 180,E1 -29488.516,E2 -29488.516} C_VEL
LIN {X 0,Y 100.97,Z 631.723,A -85,B 0,C 180,E1 -29492.555,E2 -29492.555} C_VEL
LIN {X 0,Y 112.085,Z 621.157,A -85,B 0,C 180,E1 -29495.392,E2 -29495.392} C_VEL
LIN {X 0,Y 123.38,Z 608.777,A -85,B 0,C 180,E1 -29497.764,E2 -29497.764} C_VEL
LIN {X 0,Y 133.17,Z 596.335,A -85,B 0,C 180,E1 -29499.512,E2 -29499.512} C_VEL
LIN {X 0,Y 142.27,Z 582.86,A -85,B 0,C 180,E1 -29500.865,E2 -29500.865} C_VEL
LIN {X 0,Y 149.695,Z 569.79,A -85,B 0,C 180,E1 -29501.936,E2 -29501.936} C_VEL
LIN {X 0,Y 156.331,Z 556.09,A -85,B 0,C 180,E1 -29502.806,E2 -29502.806} C_VEL
LIN {X 0,Y 162.614,Z 540.268,A -85,B 0,C 180,E1 -29503.519,E2 -29503.519} C_VEL
LIN {X 0,Y 167.639,Z 523.759,A -85,B 0,C 180,E1 -29504.074,E2 -29504.074} C_VEL
LIN {X 0,Y 171.209,Z 507.634,A -85,B 0,C 180,E1 -29504.428,E2 -29504.428} C_VEL
LIN {X 0,Y 174.28,Z 485.615,A -85,B 0,C 180,E1 -29504.794,E2 -29504.794} C_VEL
LIN {X 0,Y 176.54,Z 466.349,A -85,B 0,C 180,E1 -29505.162,E2 -29505.162} C_VEL
LIN {X 0,Y 175.907,Z 463.811,A -85,B 0,C 180,E1 -29507.809,E2 -29507.809} C_VEL
LIN {X 0,Y 175.597,Z 462.451,A -85,B 0,C 180,E1 -29509.887,E2 -29509.887} C_VEL
LIN {X 0,Y 175.44,Z 461.387,A -85,B 0,C 180,E1 -29513.096,E2 -29513.096} C_VEL
LIN {X 0,Y 175.581,Z 461.65,A -85,B 0,C 180,E1 -29515.988,E2 -29515.988} C_VEL
LIN {X 0,Y 175.839,Z 462.937,A -85,B 0,C 180,E1 -29518.152,E2 -29518.152} C_VEL
LIN {X 0,Y 176.431,Z 465.663,A -85,B 0,C 180,E1 -29520.986,E2 -29520.986} C_VEL
LIN {X 0,Y 176.581,Z 466.521,A -85,B 0,C 180,E1 -29521.593,E2 -29521.593} C_VEL
LIN {X 0,Y 171.72,Z 505.71,A -85,B 0,C 180,E1 -29522.248,E2 -29522.248} C_VEL
LIN {X 0,Y 167.967,Z 523.571,A -85,B 0,C 180,E1 -29522.61,E2 -29522.61} C_VEL
LIN {X 0,Y 163.193,Z 539.538,A -85,B 0,C 180,E1 -29523.054,E2 -29523.054} C_VEL
LIN {X 0,Y 157.123,Z 555.265,A -85,B 0,C 180,E1 -29523.608,E2 -29523.608} C_VEL
LIN {X 0,Y 149.792,Z 570.685,A -85,B 0,C 180,E1 -29524.432,E2 -29524.432} C_VEL
LIN {X 0,Y 142.057,Z 584.266,A -85,B 0,C 180,E1 -29525.351,E2 -29525.351} C_VEL
LIN {X 0,Y 133.507,Z 596.933,A -85,B 0,C 180,E1 -29526.485,E2 -29526.485} C_VEL
LIN {X 0,Y 124.196,Z 608.958,A -85,B 0,C 180,E1 -29527.994,E2 -29527.994} C_VEL
LIN {X 0,Y 114.143,Z 620.302,A -85,B 0,C 180,E1 -29529.889,E2 -29529.889} C_VEL
LIN {X 0,Y 102.616,Z 631.535,A -85,B 0,C 180,E1 -29532.592,E2 -29532.592} C_VEL
LIN {X 0,Y 91.356,Z 641.122,A -85,B 0,C 180,E1 -29535.926,E2 -29535.926} C_VEL
LIN {X 0,Y 78.783,Z 650.531,A -85,B 0,C 180,E1 -29540.903,E2 -29540.903} C_VEL
LIN {X 0,Y 67.369,Z 658.192,A -85,B 0,C 180,E1 -29547.537,E2 -29547.537} C_VEL
LIN {X 0,Y 56.989,Z 664.504,A -85,B 0,C 180,E1 -29556.719,E2 -29556.719} C_VEL
LIN {X 0,Y 48.534,Z 669.623,A -85,B 0,C 180,E1 -29569.337,E2 -29569.337} C_VEL
LIN {X 0,Y 42.13,Z 674.404,A -85,B 0,C 180,E1 -29590.512,E2 -29590.512} C_VEL
LIN {X 0,Y 41.246,Z 675.87,A -85,B 0,C 180,E1 -29600.19,E2 -29600.19} C_VEL
LIN {X 0,Y 41.306,Z 677.003,A -85,B 0,C 180,E1 -29610.001,E2 -29610.001} C_VEL
LIN {X 0,Y 42.203,Z 678.475,A -85,B 0,C 180,E1 -29629.456,E2 -29629.456} C_VEL
LIN {X 0,Y 46.995,Z 678.998,A -85,B 0,C 180,E1 -29646.742,E2 -29646.742} C_VEL
LIN {X 0,Y 55.774,Z 678.524,A -85,B 0,C 180,E1 -29660.951,E2 -29660.951} C_VEL
LIN {X 0,Y 65.163,Z 677.279,A -85,B 0,C 180,E1 -29669.637,E2 -29669.637} C_VEL
LIN {X 0,Y 76.597,Z 675.057,A -85,B 0,C 180,E1 -29676.57,E2 -29676.57} C_VEL
LIN {X 0,Y 88.871,Z 671.825,A -85,B 0,C 180,E1 -29681.619,E2 -29681.619} C_VEL
LIN {X 0,Y 101.683,Z 667.634,A -85,B 0,C 180,E1 -29685.385,E2 -29685.385} C_VEL
LIN {X 0,Y 114.854,Z 662.332,A -85,B 0,C 180,E1 -29688.254,E2 -29688.254} C_VEL
LIN {X 0,Y 128.242,Z 655.885,A -85,B 0,C 180,E1 -29690.559,E2 -29690.559} C_VEL
LIN {X 0,Y 141.821,Z 648.198,A -85,B 0,C 180,E1 -29692.357,E2 -29692.357} C_VEL
LIN {X 0,Y 155.525,Z 638.959,A -85,B 0,C 180,E1 -29693.804,E2 -29693.804} C_VEL
LIN {X 0,Y 157.641,Z 637.441,A -85,B 0,C 180,E1 -29693.99,E2 -29693.99} C_VEL
LIN {X 0,Y 158.518,Z 636.743,A -85,B 0,C 180,E1 -29694.375,E2 -29694.375} C_VEL
LIN {X 0,Y 144.436,Z 646.335,A -85,B 0,C 180,E1 -29695.947,E2 -29695.947} C_VEL
LIN {X 0,Y 130.172,Z 654.504,A -85,B 0,C 180,E1 -29697.944,E2 -29697.944} C_VEL
LIN {X 0,Y 124.985,Z 657.154,A -85,B 0,C 180,E1 -29698.448,E2 -29698.448} C_VEL
LIN {X 0,Y 108.611,Z 664.238,A -85,B 0,C 180,E1 -29698.637,E2 -29698.637} C_VEL
LIN {X 0,Y 103.145,Z 666.211,A -85,B 0,C 180,E1 -29699.146,E2 -29699.146} C_VEL
LIN {X 0,Y 101.375,Z 666.821,A -85,B 0,C 180,E1 -29699.475,E2 -29699.475} C_VEL
LIN {X 0,Y 91.414,Z 669.984,A -85,B 0,C 180,E1 -29701.886,E2 -29701.886} C_VEL
LIN {X 0,Y 77.783,Z 673.349,A -85,B 0,C 180,E1 -29706.327,E2 -29706.327} C_VEL
LIN {X 0,Y 64.585,Z 675.709,A -85,B 0,C 180,E1 -29712.574,E2 -29712.574} C_VEL
LIN {X 0,Y 52.829,Z 676.933,A -85,B 0,C 180,E1 -29721.371,E2 -29721.371} C_VEL
LIN {X 0,Y 42.722,Z 677.166,A -85,B 0,C 180,E1 -29734.66,E2 -29734.66} C_VEL
LIN {X 0,Y 35.887,Z 676.395,A -85,B 0,C 180,E1 -29754.018,E2 -29754.018} C_VEL
LIN {X 0,Y 33.522,Z 674.609,A -85,B 0,C 180,E1 -29777.897,E2 -29777.897} C_VEL
LIN {X 0,Y 35.365,Z 672.534,A -85,B 0,C 180,E1 -29796.408,E2 -29796.408} C_VEL
LIN {X 0,Y 40.527,Z 669.192,A -85,B 0,C 180,E1 -29815.691,E2 -29815.691} C_VEL
LIN {X 0,Y 49.033,Z 664.636,A -85,B 0,C 180,E1 -29830.164,E2 -29830.164} C_VEL
LIN {X 0,Y 59.466,Z 658.996,A -85,B 0,C 180,E1 -29840.192,E2 -29840.192} C_VEL
LIN {X 0,Y 71.18,Z 652.128,A -85,B 0,C 180,E1 -29847.061,E2 -29847.061} C_VEL
LIN {X 0,Y 83.525,Z 643.799,A -85,B 0,C 180,E1 -29852.066,E2 -29852.066} C_VEL
LIN {X 0,Y 96.303,Z 633.902,A -85,B 0,C 180,E1 -29855.813,E2 -29855.813} C_VEL
LIN {X 0,Y 107.706,Z 623.729,A -85,B 0,C 180,E1 -29858.408,E2 -29858.408} C_VEL
LIN {X 0,Y 119.232,Z 611.817,A -85,B 0,C 180,E1 -29860.578,E2 -29860.578} C_VEL
LIN {X 0,Y 130.021,Z 598.703,A -85,B 0,C 180,E1 -29862.302,E2 -29862.302} C_VEL
LIN {X 0,Y 139.257,Z 585.558,A -85,B 0,C 180,E1 -29863.512,E2 -29863.512} C_VEL
LIN {X 0,Y 147.672,Z 571.451,A -85,B 0,C 180,E1 -29864.522,E2 -29864.522} C_VEL
LIN {X 0,Y 154.399,Z 558.093,A -85,B 0,C 180,E1 -29865.298,E2 -29865.298} C_VEL
LIN {X 0,Y 160.763,Z 542.574,A -85,B 0,C 180,E1 -29865.919,E2 -29865.919} C_VEL
LIN {X 0,Y 166.063,Z 526.018,A -85,B 0,C 180,E1 -29866.425,E2 -29866.425} C_VEL
LIN {X 0,Y 169.876,Z 509.812,A -85,B 0,C 180,E1 -29866.763,E2 -29866.763} C_VEL
LIN {X 0,Y 172.525,Z 492.815,A -85,B 0,C 180,E1 -29867.006,E2 -29867.006} C_VEL
LIN {X 0,Y 175.087,Z 471.402,A -85,B 0,C 180,E1 -29867.374,E2 -29867.374} C_VEL
LIN {X 0,Y 174.725,Z 469.525,A -85,B 0,C 180,E1 -29869.836,E2 -29869.836} C_VEL
LIN {X 0,Y 174.559,Z 468.48,A -85,B 0,C 180,E1 -29873.061,E2 -29873.061} C_VEL
LIN {X 0,Y 174.695,Z 468.733,A -85,B 0,C 180,E1 -29875.962,E2 -29875.962} C_VEL
LIN {X 0,Y 174.884,Z 469.951,A -85,B 0,C 180,E1 -29877.82,E2 -29877.82} C_VEL
LIN {X 0,Y 175.138,Z 471.259,A -85,B 0,C 180,E1 -29879.344,E2 -29879.344} C_VEL
LIN {X 0,Y 170.675,Z 506.202,A -85,B 0,C 180,E1 -29879.905,E2 -29879.905} C_VEL
LIN {X 0,Y 166.916,Z 523.743,A -85,B 0,C 180,E1 -29880.213,E2 -29880.213} C_VEL
LIN {X 0,Y 161.652,Z 540.907,A -85,B 0,C 180,E1 -29880.584,E2 -29880.584} C_VEL
LIN {X 0,Y 155.959,Z 555.283,A -85,B 0,C 180,E1 -29881.051,E2 -29881.051} C_VEL
LIN {X 0,Y 148.535,Z 570.655,A -85,B 0,C 180,E1 -29881.749,E2 -29881.749} C_VEL
LIN {X 0,Y 140.697,Z 584.208,A -85,B 0,C 180,E1 -29882.534,E2 -29882.534} C_VEL
LIN {X 0,Y 132.019,Z 596.857,A -85,B 0,C 180,E1 -29883.488,E2 -29883.488} C_VEL
LIN {X 0,Y 123.4,Z 607.867,A -85,B 0,C 180,E1 -29884.678,E2 -29884.678} C_VEL
LIN {X 0,Y 113.122,Z 619.286,A -85,B 0,C 180,E1 -29886.26,E2 -29886.26} C_VEL
LIN {X 0,Y 101.132,Z 630.792,A -85,B 0,C 180,E1 -29888.63,E2 -29888.63} C_VEL
LIN {X 0,Y 89.633,Z 640.349,A -85,B 0,C 180,E1 -29891.451,E2 -29891.451} C_VEL
LIN {X 0,Y 76.96,Z 649.567,A -85,B 0,C 180,E1 -29895.659,E2 -29895.659} C_VEL
LIN {X 0,Y 64.343,Z 657.58,A -85,B 0,C 180,E1 -29901.811,E2 -29901.811} C_VEL
LIN {X 0,Y 52.978,Z 663.971,A -85,B 0,C 180,E1 -29910.429,E2 -29910.429} C_VEL
LIN {X 0,Y 43.317,Z 669.172,A -85,B 0,C 180,E1 -29923.107,E2 -29923.107} C_VEL
LIN {X 0,Y 37.846,Z 672.276,A -85,B 0,C 180,E1 -29936.146,E2 -29936.146} C_VEL
LIN {X 0,Y 34.218,Z 675.509,A -85,B 0,C 180,E1 -29958.149,E2 -29958.149} C_VEL
LIN {X 0,Y 34.178,Z 676.67,A -85,B 0,C 180,E1 -29970.001,E2 -29970.001} C_VEL
LIN {X 0,Y 35.533,Z 678.212,A -85,B 0,C 180,E1 -29993.303,E2 -29993.303} C_VEL
LIN {X 0,Y 41.465,Z 678.77,A -85,B 0,C 180,E1 -30012.687,E2 -30012.687} C_VEL
LIN {X 0,Y 50.811,Z 678.442,A -85,B 0,C 180,E1 -30026.414,E2 -30026.414} C_VEL
LIN {X 0,Y 61.842,Z 677.159,A -85,B 0,C 180,E1 -30035.392,E2 -30035.392} C_VEL
LIN {X 0,Y 74.034,Z 675.009,A -85,B 0,C 180,E1 -30041.678,E2 -30041.678} C_VEL
LIN {X 0,Y 86.873,Z 671.816,A -85,B 0,C 180,E1 -30046.122,E2 -30046.122} C_VEL
LIN {X 0,Y 103.467,Z 666.458,A -85,B 0,C 180,E1 -30050.039,E2 -30050.039} C_VEL
LIN {X 0,Y 117.012,Z 661.006,A -85,B 0,C 180,E1 -30052.321,E2 -30052.321} C_VEL
LIN {X 0,Y 129.21,Z 655.06,A -85,B 0,C 180,E1 -30053.966,E2 -30053.966} C_VEL
LIN {X 0,Y 131.067,Z 654.068,A -85,B 0,C 180,E1 -30054.594,E2 -30054.594} C_VEL
LIN {X 0,Y 116.916,Z 660.852,A -85,B 0,C 180,E1 -30056.556,E2 -30056.556} C_VEL
LIN {X 0,Y 101.375,Z 666.821,A -85,B 0,C 180,E1 -30059.475,E2 -30059.475} C_VEL
LIN {X 0,Y 95.917,Z 668.599,A -85,B 0,C 180,E1 -30060.306,E2 -30060.306} C_VEL
LIN {X 0,Y 86.388,Z 671.275,A -85,B 0,C 180,E1 -30060.793,E2 -30060.793} C_VEL
LIN {X 0,Y 78.675,Z 673.104,A -85,B 0,C 180,E1 -30061.196,E2 -30061.196} C_VEL
LIN {X 0,Y 73.024,Z 674.284,A -85,B 0,C 180,E1 -30062.165,E2 -30062.165} C_VEL
LIN {X 0,Y 71.22,Z 674.56,A -85,B 0,C 180,E1 -30062.724,E2 -30062.724} C_VEL
LIN {X 0,Y 56.951,Z 676.585,A -85,B 0,C 180,E1 -30069.159,E2 -30069.159} C_VEL
LIN {X 0,Y 44.526,Z 677.366,A -85,B 0,C 180,E1 -30078.728,E2 -30078.728} C_VEL
LIN {X 0,Y 34.067,Z 677.191,A -85,B 0,C 180,E1 -30094.388,E2 -30094.388} C_VEL
LIN {X 0,Y 27.522,Z 675.926,A -85,B 0,C 180,E1 -30119.286,E2 -30119.286} C_VEL
LIN {X 0,Y 27.045,Z 673.764,A -85,B 0,C 180,E1 -30149.998,E2 -30149.998} C_VEL
LIN {X 0,Y 29.239,Z 672.268,A -85,B 0,C 180,E1 -30163.906,E2 -30163.906} C_VEL
LIN {X 0,Y 36.41,Z 668.58,A -85,B 0,C 180,E1 -30185.383,E2 -30185.383} C_VEL
LIN {X 0,Y 46.566,Z 663.893,A -85,B 0,C 180,E1 -30198.992,E2 -30198.992} C_VEL
LIN {X 0,Y 61.301,Z 656.357,A -85,B 0,C 180,E1 -30209.299,E2 -30209.299} C_VEL
LIN {X 0,Y 75.597,Z 647.812,A -85,B 0,C 180,E1 -30215.015,E2 -30215.015} C_VEL
LIN {X 0,Y 88.667,Z 638.614,A -85,B 0,C 180,E1 -30218.643,E2 -30218.643} C_VEL
LIN {X 0,Y 100.29,Z 629.165,A -85,B 0,C 180,E1 -30221.09,E2 -30221.09} C_VEL
LIN {X 0,Y 112.015,Z 618.174,A -85,B 0,C 180,E1 -30223.098,E2 -30223.098} C_VEL
LIN {X 0,Y 123.831,Z 605.181,A -85,B 0,C 180,E1 -30224.759,E2 -30224.759} C_VEL
LIN {X 0,Y 134.018,Z 591.931,A -85,B 0,C 180,E1 -30225.964,E2 -30225.964} C_VEL
LIN {X 0,Y 142.537,Z 578.926,A -85,B 0,C 180,E1 -30226.855,E2 -30226.855} C_VEL
LIN {X 0,Y 150.195,Z 565.185,A -85,B 0,C 180,E1 -30227.632,E2 -30227.632} C_VEL
LIN {X 0,Y 157.486,Z 549.32,A -85,B 0,C 180,E1 -30228.233,E2 -30228.233} C_VEL
LIN {X 0,Y 163.487,Z 532.64,A -85,B 0,C 180,E1 -30228.713,E2 -30228.713} C_VEL
LIN {X 0,Y 167.892,Z 516.255,A -85,B 0,C 180,E1 -30229.052,E2 -30229.052} C_VEL
LIN {X 0,Y 170.87,Z 500.387,A -85,B 0,C 180,E1 -30229.262,E2 -30229.262} C_VEL
LIN {X 0,Y 173.842,Z 476.949,A -85,B 0,C 180,E1 -30229.604,E2 -30229.604} C_VEL
